LIN {X 0,Y 411.455,Z 725.231,A -85,B 0,C 180,E1 -10613.133,E2 -10613.133} C_VEL
LIN {X 0,Y 411.306,Z 725.25,A -85,B 0,C 180,E1 -10615.099,E2 -10615.099} C_VEL
LIN {X 0,Y 411.51,Z 725.225,A -85,B 0,C 180,E1 -10618.043,E2 -10618.043} C_VEL
LIN {X 0,Y 411.638,Z 725.209,A -85,B 0,C 180,E1 -10620,E2 -10620} C_VEL
LIN {X 0,Y 411.452,Z 725.232,A -85,B 0,C 180,E1 -10622.937,E2 -10622.937} C_VEL
LIN {X 0,Y 411.425,Z 725.236,A -85,B 0,C 180,E1 -10626.868,E2 -10626.868} C_VEL
LIN {X 0,Y 411.293,Z 725.251,A -85,B 0,C 180,E1 -10629.839,E2 -10629.839} C_VEL
LIN {X 0,Y 411.308,Z 725.25,A -85,B 0,C 180,E1 -10633.104,E2 -10633.104} C_VEL
LIN {X 0,Y 411.259,Z 725.258,A -85,B 0,C 180,E1 -10636.889,E2 -10636.889} C_VEL
LIN {X 0,Y 411.233,Z 725.259,A -85,B 0,C 180,E1 -10639.987,E2 -10639.987} C_VEL
LIN {X 0,Y 411.189,Z 725.266,A -85,B 0,C 180,E1 -10643.149,E2 -10643.149} C_VEL
LIN {X 0,Y 411.186,Z 725.265,A -85,B 0,C 180,E1 -10646.385,E2 -10646.385} C_VEL
LIN {X 0,Y 411.2,Z 725.264,A -85,B 0,C 180,E1 -10649.713,E2 -10649.713} C_VEL
LIN {X 0,Y 411.206,Z 725.265,A -85,B 0,C 180,E1 -10653.156,E2 -10653.156} C_VEL
LIN {X 0,Y 411.192,Z 725.264,A -85,B 0,C 180,E1 -10656.552,E2 -10656.552} C_VEL
LIN {X 0,Y 411.169,Z 725.268,A -85,B 0,C 180,E1 -10659.72,E2 -10659.72} C_VEL
LIN {X 0,Y 411.164,Z 725.268,A -85,B 0,C 180,E1 -10663.135,E2 -10663.135} C_VEL
LIN {X 0,Y 411.165,Z 725.268,A -85,B 0,C 180,E1 -10665.882,E2 -10665.882} C_VEL
LIN {X 0,Y 411.149,Z 725.27,A -85,B 0,C 180,E1 -10668.775,E2 -10668.775} C_VEL
LIN {X 0,Y 411.183,Z 725.266,A -85,B 0,C 180,E1 -10672.025,E2 -10672.025} C_VEL
LIN {X 0,Y 411.202,Z 725.263,A -85,B 0,C 180,E1 -10675.124,E2 -10675.124} C_VEL
LIN {X 0,Y 411.156,Z 725.269,A -85,B 0,C 180,E1 -10678.002,E2 -10678.002} C_VEL
LIN {X 0,Y 411.171,Z 725.267,A -85,B 0,C 180,E1 -10681.406,E2 -10681.406} C_VEL
LIN {X 0,Y 411.189,Z 725.267,A -85,B 0,C 180,E1 -10684.942,E2 -10684.942} C_VEL
LIN {X 0,Y 411.206,Z 725.263,A -85,B 0,C 180,E1 -10687.913,E2 -10687.913} C_VEL
LIN {X 0,Y 411.221,Z 725.263,A -85,B 0,C 180,E1 -10691.051,E2 -10691.051} C_VEL
LIN {X 0,Y 411.253,Z 725.258,A -85,B 0,C 180,E1 -10694.132,E2 -10694.132} C_VEL
LIN {X 0,Y 411.305,Z 725.253,A -85,B 0,C 180,E1 -10697.166,E2 -10697.166} C_VEL
LIN {X 0,Y 411.276,Z 725.254,A -85,B 0,C 180,E1 -10700.161,E2 -10700.161} C_VEL
LIN {X 0,Y 411.393,Z 725.242,A -85,B 0,C 180,E1 -10703.132,E2 -10703.132} C_VEL
LIN {X 0,Y 411.287,Z 725.254,A -85,B 0,C 180,E1 -10705.099,E2 -10705.099} C_VEL
LIN {X 0,Y 411.504,Z 725.224,A -85,B 0,C 180,E1 -10708.043,E2 -10708.043} C_VEL
LIN {X 0,Y 411.38,Z 725.241,A -85,B 0,C 180,E1 -10710.979,E2 -10710.979} C_VEL
LIN {X 0,Y 411.432,Z 725.234,A -85,B 0,C 180,E1 -10712.938,E2 -10712.938} C_VEL
LIN {X 0,Y 411.432,Z 725.235,A -85,B 0,C 180,E1 -10715.883,E2 -10715.883} C_VEL
LIN {X 0,Y 411.32,Z 725.247,A -85,B 0,C 180,E1 -10718.846,E2 -10718.846} C_VEL
LIN {X 0,Y 411.286,Z 725.255,A -85,B 0,C 180,E1 -10721.833,E2 -10721.833} C_VEL
LIN {X 0,Y 411.263,Z 725.254,A -85,B 0,C 180,E1 -10724.853,E2 -10724.853} C_VEL
LIN {X 0,Y 411.241,Z 725.258,A -85,B 0,C 180,E1 -10727.571,E2 -10727.571} C_VEL
LIN {X 0,Y 410.579,Z 725.344,A -85,B 0,C 180,E1 -10728.389,E2 -10728.389} C_VEL
LIN {X 0,Y 407.693,Z 725.704,A -85,B 0,C 180,E1 -10729.717,E2 -10729.717} C_VEL
LIN {X 0,Y 405.251,Z 726.005,A -85,B 0,C 180,E1 -10730.79,E2 -10730.79} C_VEL
LIN {X 0,Y 404.215,Z 726.134,A -85,B 0,C 180,E1 -10731.62,E2 -10731.62} C_VEL
LIN {X 0,Y 404.138,Z 726.14,A -85,B 0,C 180,E1 -10731.901,E2 -10731.901} C_VEL
LIN {X 0,Y 404.155,Z 726.139,A -85,B 0,C 180,E1 -10735.277,E2 -10735.277} C_VEL
LIN {X 0,Y 404.133,Z 726.147,A -85,B 0,C 180,E1 -10738.005,E2 -10738.005} C_VEL
LIN {X 0,Y 404.148,Z 726.143,A -85,B 0,C 180,E1 -10740.285,E2 -10740.285} C_VEL
LIN {X 0,Y 404.148,Z 726.142,A -85,B 0,C 180,E1 -10743.812,E2 -10743.812} C_VEL
LIN {X 0,Y 404.139,Z 726.141,A -85,B 0,C 180,E1 -10746.875,E2 -10746.875} C_VEL
LIN {X 0,Y 404.151,Z 726.142,A -85,B 0,C 180,E1 -10750.08,E2 -10750.08} C_VEL
LIN {X 0,Y 404.156,Z 726.139,A -85,B 0,C 180,E1 -10753.084,E2 -10753.084} C_VEL
LIN {X 0,Y 404.158,Z 726.14,A -85,B 0,C 180,E1 -10755.411,E2 -10755.411} C_VEL
LIN {X 0,Y 407.371,Z 737.515,A -85,B 0,C 180,E1 -10756.25,E2 -10756.25} C_VEL
LIN {X 0,Y 408.302,Z 740.837,A -85,B 0,C 180,E1 -10756.535,E2 -10756.535} C_VEL
LIN {X 0,Y 407.909,Z 751.917,A -85,B 0,C 180,E1 -10757.448,E2 -10757.448} C_VEL
LIN {X 0,Y 407.285,Z 762.487,A -85,B 0,C 180,E1 -10758.533,E2 -10758.533} C_VEL
LIN {X 0,Y 406.729,Z 771.783,A -85,B 0,C 180,E1 -10759.703,E2 -10759.703} C_VEL
LIN {X 0,Y 406.09,Z 781.183,A -85,B 0,C 180,E1 -10761.151,E2 -10761.151} C_VEL
LIN {X 0,Y 405.509,Z 789.001,A -85,B 0,C 180,E1 -10762.656,E2 -10762.656} C_VEL
LIN {X 0,Y 405.021,Z 795.844,A -85,B 0,C 180,E1 -10764.311,E2 -10764.311} C_VEL
LIN {X 0,Y 404.679,Z 800.21,A -85,B 0,C 180,E1 -10765.637,E2 -10765.637} C_VEL
LIN {X 0,Y 404.479,Z 804.684,A -85,B 0,C 180,E1 -10767.409,E2 -10767.409} C_VEL
LIN {X 0,Y 404.335,Z 806.818,A -85,B 0,C 180,E1 -10768.57,E2 -10768.57} C_VEL
LIN {X 0,Y 404.169,Z 809.071,A -85,B 0,C 180,E1 -10770.394,E2 -10770.394} C_VEL
LIN {X 0,Y 404.199,Z 809.968,A -85,B 0,C 180,E1 -10772.47,E2 -10772.47} C_VEL
LIN {X 0,Y 404.33,Z 809.377,A -85,B 0,C 180,E1 -10774.243,E2 -10774.243} C_VEL
LIN {X 0,Y 404.513,Z 808.375,A -85,B 0,C 180,E1 -10775.356,E2 -10775.356} C_VEL
LIN {X 0,Y 404.79,Z 806.008,A -85,B 0,C 180,E1 -10776.955,E2 -10776.955} C_VEL
LIN {X 0,Y 405.183,Z 802.282,A -85,B 0,C 180,E1 -10778.638,E2 -10778.638} C_VEL
LIN {X 0,Y 405.666,Z 797.413,A -85,B 0,C 180,E1 -10780.255,E2 -10780.255} C_VEL
LIN {X 0,Y 406.317,Z 791.148,A -85,B 0,C 180,E1 -10781.86,E2 -10781.86} C_VEL
LIN {X 0,Y 407.106,Z 783.159,A -85,B 0,C 180,E1 -10783.45,E2 -10783.45} C_VEL
LIN {X 0,Y 407.851,Z 774.76,A -85,B 0,C 180,E1 -10784.793,E2 -10784.793} C_VEL
LIN {X 0,Y 408.577,Z 764.958,A -85,B 0,C 180,E1 -10786.065,E2 -10786.065} C_VEL
LIN {X 0,Y 409.312,Z 753.636,A -85,B 0,C 180,E1 -10787.228,E2 -10787.228} C_VEL
LIN {X 0,Y 409.772,Z 744.554,A -85,B 0,C 180,E1 -10787.985,E2 -10787.985} C_VEL
LIN {X 0,Y 408.712,Z 739.651,A -85,B 0,C 180,E1 -10788.411,E2 -10788.411} C_VEL
LIN {X 0,Y 404.722,Z 727.908,A -85,B 0,C 180,E1 -10789.368,E2 -10789.368} C_VEL
LIN {X 0,Y 404.259,Z 726.133,A -85,B 0,C 180,E1 -10789.514,E2 -10789.514} C_VEL
LIN {X 0,Y 404.363,Z 726.114,A -85,B 0,C 180,E1 -10793.012,E2 -10793.012} C_VEL
LIN {X 0,Y 404.277,Z 726.124,A -85,B 0,C 180,E1 -10795.013,E2 -10795.013} C_VEL
LIN {X 0,Y 404.482,Z 726.104,A -85,B 0,C 180,E1 -10798.008,E2 -10798.008} C_VEL
LIN {X 0,Y 404.609,Z 726.087,A -85,B 0,C 180,E1 -10800,E2 -10800} C_VEL
LIN {X 0,Y 404.412,Z 726.103,A -85,B 0,C 180,E1 -10802.988,E2 -10802.988} C_VEL
LIN {X 0,Y 404.42,Z 726.105,A -85,B 0,C 180,E1 -10805.985,E2 -10805.985} C_VEL
LIN {X 0,Y 404.386,Z 726.112,A -85,B 0,C 180,E1 -10807.992,E2 -10807.992} C_VEL
LIN {X 0,Y 404.26,Z 726.125,A -85,B 0,C 180,E1 -10812.041,E2 -10812.041} C_VEL
LIN {X 0,Y 404.21,Z 726.127,A -85,B 0,C 180,E1 -10815.118,E2 -10815.118} C_VEL
LIN {X 0,Y 404.212,Z 726.132,A -85,B 0,C 180,E1 -10818.238,E2 -10818.238} C_VEL
LIN {X 0,Y 404.142,Z 726.137,A -85,B 0,C 180,E1 -10821.419,E2 -10821.419} C_VEL
LIN {X 0,Y 404.177,Z 726.14,A -85,B 0,C 180,E1 -10824.666,E2 -10824.666} C_VEL
LIN {X 0,Y 404.198,Z 726.138,A -85,B 0,C 180,E1 -10827.999,E2 -10827.999} C_VEL
LIN {X 0,Y 404.142,Z 726.141,A -85,B 0,C 180,E1 -10831.558,E2 -10831.558} C_VEL
LIN {X 0,Y 404.188,Z 726.138,A -85,B 0,C 180,E1 -10835.016,E2 -10835.016} C_VEL
LIN {X 0,Y 404.159,Z 726.145,A -85,B 0,C 180,E1 -10838.757,E2 -10838.757} C_VEL
LIN {X 0,Y 404.126,Z 726.148,A -85,B 0,C 180,E1 -10841.6,E2 -10841.6} C_VEL
LIN {X 0,Y 404.148,Z 726.144,A -85,B 0,C 180,E1 -10844.522,E2 -10844.522} C_VEL
LIN {X 0,Y 404.151,Z 726.237,A -85,B 0,C 180,E1 -10845.926,E2 -10845.926} C_VEL
LIN {X 0,Y 405.706,Z 733.429,A -85,B 0,C 180,E1 -10848.832,E2 -10848.832} C_VEL
LIN {X 0,Y 407.377,Z 742.456,A -85,B 0,C 180,E1 -10852.104,E2 -10852.104} C_VEL
LIN {X 0,Y 407.587,Z 746.68,A -85,B 0,C 180,E1 -10853.495,E2 -10853.495} C_VEL
LIN {X 0,Y 406.594,Z 758.282,A -85,B 0,C 180,E1 -10857.011,E2 -10857.011} C_VEL
LIN {X 0,Y 405.823,Z 768.597,A -85,B 0,C 180,E1 -10859.985,E2 -10859.985} C_VEL
LIN {X 0,Y 405.143,Z 781.14,A -85,B 0,C 180,E1 -10863.469,E2 -10863.469} C_VEL
LIN {X 0,Y 404.529,Z 794.458,A -85,B 0,C 180,E1 -10867.041,E2 -10867.041} C_VEL
LIN {X 0,Y 404.045,Z 806.932,A -85,B 0,C 180,E1 -10870.307,E2 -10870.307} C_VEL
LIN {X 0,Y 403.943,Z 812.973,A -85,B 0,C 180,E1 -10871.875,E2 -10871.875} C_VEL
LIN {X 0,Y 405.529,Z 827.395,A -85,B 0,C 180,E1 -10872.398,E2 -10872.398} C_VEL
LIN {X 0,Y 406.374,Z 841.524,A -85,B 0,C 180,E1 -10873.096,E2 -10873.096} C_VEL
LIN {X 0,Y 407.137,Z 852.896,A -85,B 0,C 180,E1 -10873.838,E2 -10873.838} C_VEL
LIN {X 0,Y 406.352,Z 864.193,A -85,B 0,C 180,E1 -10874.707,E2 -10874.707} C_VEL
LIN {X 0,Y 405.48,Z 875.869,A -85,B 0,C 180,E1 -10875.829,E2 -10875.829} C_VEL
LIN {X 0,Y 404.907,Z 885.404,A -85,B 0,C 180,E1 -10876.959,E2 -10876.959} C_VEL
LIN {X 0,Y 404.285,Z 894.164,A -85,B 0,C 180,E1 -10878.214,E2 -10878.214} C_VEL
LIN {X 0,Y 403.775,Z 902.798,A -85,B 0,C 180,E1 -10879.723,E2 -10879.723} C_VEL
LIN {X 0,Y 403.516,Z 909.827,A -85,B 0,C 180,E1 -10881.234,E2 -10881.234} C_VEL
LIN {X 0,Y 403.398,Z 916.317,A -85,B 0,C 180,E1 -10882.995,E2 -10882.995} C_VEL
LIN {X 0,Y 403.398,Z 920.58,A -85,B 0,C 180,E1 -10884.501,E2 -10884.501} C_VEL
LIN {X 0,Y 403.532,Z 923.776,A -85,B 0,C 180,E1 -10886.005,E2 -10886.005} C_VEL
LIN {X 0,Y 403.475,Z 926.402,A -85,B 0,C 180,E1 -10888.003,E2 -10888.003} C_VEL
LIN {X 0,Y 403.481,Z 927.104,A -85,B 0,C 180,E1 -10889.002,E2 -10889.002} C_VEL
LIN {X 0,Y 403.49,Z 927.365,A -85,B 0,C 180,E1 -10890,E2 -10890} C_VEL
LIN {X 0,Y 403.472,Z 927.18,A -85,B 0,C 180,E1 -10890.998,E2 -10890.998} C_VEL
LIN {X 0,Y 403.456,Z 926.592,A -85,B 0,C 180,E1 -10891.996,E2 -10891.996} C_VEL
LIN {X 0,Y 403.445,Z 925.596,A -85,B 0,C 180,E1 -10892.996,E2 -10892.996} C_VEL
LIN {X 0,Y 403.522,Z 924.151,A -85,B 0,C 180,E1 -10893.995,E2 -10893.995} C_VEL
LIN {X 0,Y 403.355,Z 921.099,A -85,B 0,C 180,E1 -10895.499,E2 -10895.499} C_VEL
LIN {X 0,Y 403.385,Z 916.972,A -85,B 0,C 180,E1 -10897.005,E2 -10897.005} C_VEL
LIN {X 0,Y 403.513,Z 910.613,A -85,B 0,C 180,E1 -10898.766,E2 -10898.766} C_VEL
LIN {X 0,Y 403.752,Z 903.688,A -85,B 0,C 180,E1 -10900.278,E2 -10900.278} C_VEL
LIN {X 0,Y 404.299,Z 895.087,A -85,B 0,C 180,E1 -10901.786,E2 -10901.786} C_VEL
LIN {X 0,Y 405.011,Z 886.285,A -85,B 0,C 180,E1 -10903.037,E2 -10903.037} C_VEL
LIN {X 0,Y 405.484,Z 877.813,A -85,B 0,C 180,E1 -10904.043,E2 -10904.043} C_VEL
LIN {X 0,Y 406.233,Z 866.186,A -85,B 0,C 180,E1 -10905.169,E2 -10905.169} C_VEL
LIN {X 0,Y 407.097,Z 854.815,A -85,B 0,C 180,E1 -10906.035,E2 -10906.035} C_VEL
LIN {X 0,Y 406.529,Z 845.674,A -85,B 0,C 180,E1 -10906.62,E2 -10906.62} C_VEL
LIN {X 0,Y 405.565,Z 832.566,A -85,B 0,C 180,E1 -10907.282,E2 -10907.282} C_VEL
LIN {X 0,Y 404.071,Z 818.692,A -85,B 0,C 180,E1 -10907.773,E2 -10907.773} C_VEL
LIN {X 0,Y 403.964,Z 816.966,A -85,B 0,C 180,E1 -10907.856,E2 -10907.856} C_VEL
LIN {X 0,Y 404.461,Z 803.727,A -85,B 0,C 180,E1 -10911.401,E2 -10911.401} C_VEL
LIN {X 0,Y 405.173,Z 790.061,A -85,B 0,C 180,E1 -10915.115,E2 -10915.115} C_VEL
LIN {X 0,Y 405.983,Z 778.085,A -85,B 0,C 180,E1 -10918.43,E2 -10918.43} C_VEL
LIN {X 0,Y 406.985,Z 764.176,A -85,B 0,C 180,E1 -10922.366,E2 -10922.366} C_VEL
LIN {X 0,Y 408.045,Z 752.225,A -85,B 0,C 180,E1 -10925.846,E2 -10925.846} C_VEL
LIN {X 0,Y 408.334,Z 748.205,A -85,B 0,C 180,E1 -10927.042,E2 -10927.042} C_VEL
LIN {X 0,Y 407.789,Z 744.091,A -85,B 0,C 180,E1 -10928.348,E2 -10928.348} C_VEL
LIN {X 0,Y 405.697,Z 733.602,A -85,B 0,C 180,E1 -10931.849,E2 -10931.849} C_VEL
LIN {X 0,Y 404.157,Z 726.141,A -85,B 0,C 180,E1 -10934.524,E2 -10934.524} C_VEL
LIN {X 0,Y 404.138,Z 726.145,A -85,B 0,C 180,E1 -10937.296,E2 -10937.296} C_VEL
LIN {X 0,Y 404.17,Z 726.138,A -85,B 0,C 180,E1 -10939.955,E2 -10939.955} C_VEL
LIN {X 0,Y 404.138,Z 726.142,A -85,B 0,C 180,E1 -10943.125,E2 -10943.125} C_VEL
LIN {X 0,Y 404.147,Z 726.141,A -85,B 0,C 180,E1 -10946.188,E2 -10946.188} C_VEL
LIN {X 0,Y 404.147,Z 726.146,A -85,B 0,C 180,E1 -10949.715,E2 -10949.715} C_VEL
LIN {X 0,Y 404.196,Z 726.134,A -85,B 0,C 180,E1 -10953.123,E2 -10953.123} C_VEL
LIN {X 0,Y 404.176,Z 726.137,A -85,B 0,C 180,E1 -10955.334,E2 -10955.334} C_VEL
LIN {X 0,Y 404.14,Z 726.142,A -85,B 0,C 180,E1 -10958.581,E2 -10958.581} C_VEL
LIN {X 0,Y 404.211,Z 726.135,A -85,B 0,C 180,E1 -10961.762,E2 -10961.762} C_VEL
LIN {X 0,Y 404.208,Z 726.133,A -85,B 0,C 180,E1 -10964.882,E2 -10964.882} C_VEL
LIN {X 0,Y 404.258,Z 726.13,A -85,B 0,C 180,E1 -10967.959,E2 -10967.959} C_VEL
LIN {X 0,Y 404.407,Z 726.112,A -85,B 0,C 180,E1 -10972.129,E2 -10972.129} C_VEL
LIN {X 0,Y 404.422,Z 726.108,A -85,B 0,C 180,E1 -10974.015,E2 -10974.015} C_VEL
LIN {X 0,Y 404.479,Z 726.101,A -85,B 0,C 180,E1 -10978.009,E2 -10978.009} C_VEL
LIN {X 0,Y 404.608,Z 726.084,A -85,B 0,C 180,E1 -10980,E2 -10980} C_VEL
LIN {X 0,Y 404.41,Z 726.109,A -85,B 0,C 180,E1 -10982.989,E2 -10982.989} C_VEL
LIN {X 0,Y 404.371,Z 726.115,A -85,B 0,C 180,E1 -10986.988,E2 -10986.988} C_VEL
LIN {X 0,Y 404.259,Z 726.127,A -85,B 0,C 180,E1 -10990.012,E2 -10990.012} C_VEL
LIN {X 0,Y 404.269,Z 726.127,A -85,B 0,C 180,E1 -10993.211,E2 -10993.211} C_VEL
LIN {X 0,Y 404.218,Z 726.135,A -85,B 0,C 180,E1 -10997.007,E2 -10997.007} C_VEL
LIN {X 0,Y 404.166,Z 726.139,A -85,B 0,C 180,E1 -11000.352,E2 -11000.352} C_VEL
LIN {X 0,Y 404.15,Z 726.142,A -85,B 0,C 180,E1 -11003.576,E2 -11003.576} C_VEL
LIN {X 0,Y 404.131,Z 726.145,A -85,B 0,C 180,E1 -11006.882,E2 -11006.882} C_VEL
LIN {X 0,Y 404.146,Z 726.142,A -85,B 0,C 180,E1 -11010.285,E2 -11010.285} C_VEL
LIN {X 0,Y 404.14,Z 726.144,A -85,B 0,C 180,E1 -11013.813,E2 -11013.813} C_VEL
LIN {X 0,Y 404.135,Z 726.143,A -85,B 0,C 180,E1 -11016.874,E2 -11016.874} C_VEL
LIN {X 0,Y 404.118,Z 726.147,A -85,B 0,C 180,E1 -11020.075,E2 -11020.075} C_VEL
LIN {X 0,Y 404.143,Z 726.142,A -85,B 0,C 180,E1 -11023.082,E2 -11023.082} C_VEL
LIN {X 0,Y 404.122,Z 726.146,A -85,B 0,C 180,E1 -11025.922,E2 -11025.922} C_VEL
LIN {X 0,Y 404.103,Z 726.148,A -85,B 0,C 180,E1 -11028.633,E2 -11028.633} C_VEL
LIN {X 0,Y 404.139,Z 726.144,A -85,B 0,C 180,E1 -11031.495,E2 -11031.495} C_VEL
LIN {X 0,Y 404.173,Z 726.138,A -85,B 0,C 180,E1 -11034.983,E2 -11034.983} C_VEL
LIN {X 0,Y 404.133,Z 726.145,A -85,B 0,C 180,E1 -11038.444,E2 -11038.444} C_VEL
LIN {X 0,Y 404.15,Z 726.143,A -85,B 0,C 180,E1 -11040.862,E2 -11040.862} C_VEL
LIN {X 0,Y 404.153,Z 726.143,A -85,B 0,C 180,E1 -11044.723,E2 -11044.723} C_VEL
LIN {X 0,Y 404.168,Z 726.138,A -85,B 0,C 180,E1 -11047.508,E2 -11047.508} C_VEL
LIN {X 0,Y 404.165,Z 726.141,A -85,B 0,C 180,E1 -11050.708,E2 -11050.708} C_VEL
LIN {X 0,Y 404.221,Z 726.132,A -85,B 0,C 180,E1 -11053.848,E2 -11053.848} C_VEL
LIN {X 0,Y 404.286,Z 726.127,A -85,B 0,C 180,E1 -11056.939,E2 -11056.939} C_VEL
LIN {X 0,Y 404.244,Z 726.129,A -85,B 0,C 180,E1 -11059.988,E2 -11059.988} C_VEL
LIN {X 0,Y 404.343,Z 726.119,A -85,B 0,C 180,E1 -11063.012,E2 -11063.012} C_VEL
LIN {X 0,Y 404.259,Z 726.129,A -85,B 0,C 180,E1 -11065.013,E2 -11065.013} C_VEL
LIN {X 0,Y 404.473,Z 726.1,A -85,B 0,C 180,E1 -11068.009,E2 -11068.009} C_VEL
LIN {X 0,Y 404.35,Z 726.117,A -85,B 0,C 180,E1 -11070.996,E2 -11070.996} C_VEL
LIN {X 0,Y 404.392,Z 726.112,A -85,B 0,C 180,E1 -11072.989,E2 -11072.989} C_VEL
LIN {X 0,Y 404.381,Z 726.112,A -85,B 0,C 180,E1 -11075.986,E2 -11075.986} C_VEL
LIN {X 0,Y 404.268,Z 726.126,A -85,B 0,C 180,E1 -11079.002,E2 -11079.002} C_VEL
LIN {X 0,Y 404.259,Z 726.128,A -85,B 0,C 180,E1 -11082.042,E2 -11082.042} C_VEL
LIN {X 0,Y 404.209,Z 726.133,A -85,B 0,C 180,E1 -11085.118,E2 -11085.118} C_VEL
LIN {X 0,Y 404.212,Z 726.133,A -85,B 0,C 180,E1 -11088.238,E2 -11088.238} C_VEL
LIN {X 0,Y 404.142,Z 726.142,A -85,B 0,C 180,E1 -11091.419,E2 -11091.419} C_VEL
LIN {X 0,Y 404.138,Z 726.14,A -85,B 0,C 180,E1 -11091.901,E2 -11091.901} C_VEL
LIN {X 0,Y 403.496,Z 726.222,A -85,B 0,C 180,E1 -11092.733,E2 -11092.733} C_VEL
LIN {X 0,Y 400.668,Z 726.579,A -85,B 0,C 180,E1 -11094.084,E2 -11094.084} C_VEL
LIN {X 0,Y 398.249,Z 726.883,A -85,B 0,C 180,E1 -11095.176,E2 -11095.176} C_VEL
LIN {X 0,Y 397.191,Z 727.012,A -85,B 0,C 180,E1 -11096.019,E2 -11096.019} C_VEL
LIN {X 0,Y 397.095,Z 727.021,A -85,B 0,C 180,E1 -11096.305,E2 -11096.305} C_VEL
LIN {X 0,Y 397.104,Z 727.021,A -85,B 0,C 180,E1 -11099.863,E2 -11099.863} C_VEL
LIN {X 0,Y 397.122,Z 727.016,A -85,B 0,C 180,E1 -11103.718,E2 -11103.718} C_VEL
LIN {X 0,Y 397.096,Z 727.017,A -85,B 0,C 180,E1 -11107.209,E2 -11107.209} C_VEL
LIN {X 0,Y 397.105,Z 727.022,A -85,B 0,C 180,E1 -11110.445,E2 -11110.445} C_VEL
LIN {X 0,Y 397.104,Z 727.017,A -85,B 0,C 180,E1 -11113.649,E2 -11113.649} C_VEL
LIN {X 0,Y 397.111,Z 727.023,A -85,B 0,C 180,E1 -11115.156,E2 -11115.156} C_VEL
LIN {X 0,Y 400.422,Z 738.626,A -85,B 0,C 180,E1 -11116.023,E2 -11116.023} C_VEL
LIN {X 0,Y 401.529,Z 743.37,A -85,B 0,C 180,E1 -11116.427,E2 -11116.427} C_VEL
LIN {X 0,Y 400.921,Z 754.73,A -85,B 0,C 180,E1 -11117.413,E2 -11117.413} C_VEL
LIN {X 0,Y 400.248,Z 766.257,A -85,B 0,C 180,E1 -11118.67,E2 -11118.67} C_VEL
LIN {X 0,Y 399.555,Z 776.377,A -85,B 0,C 180,E1 -11120.057,E2 -11120.057} C_VEL
LIN {X 0,Y 398.874,Z 785.472,A -85,B 0,C 180,E1 -11121.604,E2 -11121.604} C_VEL
LIN {X 0,Y 398.368,Z 792.688,A -85,B 0,C 180,E1 -11123.142,E2 -11123.142} C_VEL
LIN {X 0,Y 397.823,Z 799.388,A -85,B 0,C 180,E1 -11124.96,E2 -11124.96} C_VEL
LIN {X 0,Y 397.54,Z 804.385,A -85,B 0,C 180,E1 -11126.767,E2 -11126.767} C_VEL
LIN {X 0,Y 397.391,Z 807.1,A -85,B 0,C 180,E1 -11128.093,E2 -11128.093} C_VEL
LIN {X 0,Y 397.244,Z 808.728,A -85,B 0,C 180,E1 -11129.132,E2 -11129.132} C_VEL
LIN {X 0,Y 397.158,Z 810.018,A -85,B 0,C 180,E1 -11130.298,E2 -11130.298} C_VEL
LIN {X 0,Y 397.179,Z 811.029,A -85,B 0,C 180,E1 -11132.22,E2 -11132.22} C_VEL
LIN {X 0,Y 397.27,Z 810.791,A -85,B 0,C 180,E1 -11133.751,E2 -11133.751} C_VEL
LIN {X 0,Y 397.42,Z 810.005,A -85,B 0,C 180,E1 -11134.886,E2 -11134.886} C_VEL
LIN {X 0,Y 397.759,Z 807.642,A -85,B 0,C 180,E1 -11136.75,E2 -11136.75} C_VEL
LIN {X 0,Y 398.107,Z 804.708,A -85,B 0,C 180,E1 -11138.239,E2 -11138.239} C_VEL
LIN {X 0,Y 398.553,Z 800.302,A -85,B 0,C 180,E1 -11139.888,E2 -11139.888} C_VEL
LIN {X 0,Y 399.253,Z 794.484,A -85,B 0,C 180,E1 -11141.527,E2 -11141.527} C_VEL
LIN {X 0,Y 399.998,Z 787.113,A -85,B 0,C 180,E1 -11143.147,E2 -11143.147} C_VEL
LIN {X 0,Y 400.827,Z 778.512,A -85,B 0,C 180,E1 -11144.658,E2 -11144.658} C_VEL
LIN {X 0,Y 401.637,Z 769.297,A -85,B 0,C 180,E1 -11145.949,E2 -11145.949} C_VEL
LIN {X 0,Y 402.39,Z 758.629,A -85,B 0,C 180,E1 -11147.159,E2 -11147.159} C_VEL
LIN {X 0,Y 403.017,Z 748.139,A -85,B 0,C 180,E1 -11148.11,E2 -11148.11} C_VEL
LIN {X 0,Y 403.101,Z 745.629,A -85,B 0,C 180,E1 -11148.306,E2 -11148.306} C_VEL
LIN {X 0,Y 400.551,Z 736.775,A -85,B 0,C 180,E1 -11149.102,E2 -11149.102} C_VEL
LIN {X 0,Y 397.21,Z 727.012,A -85,B 0,C 180,E1 -11149.873,E2 -11149.873} C_VEL
LIN {X 0,Y 397.309,Z 726.993,A -85,B 0,C 180,E1 -11152.887,E2 -11152.887} C_VEL
LIN {X 0,Y 397.247,Z 727,A -85,B 0,C 180,E1 -11154.925,E2 -11154.925} C_VEL
LIN {X 0,Y 397.451,Z 726.98,A -85,B 0,C 180,E1 -11157.973,E2 -11157.973} C_VEL
LIN {X 0,Y 397.579,Z 726.962,A -85,B 0,C 180,E1 -11160,E2 -11160} C_VEL
LIN {X 0,Y 397.372,Z 726.98,A -85,B 0,C 180,E1 -11163.041,E2 -11163.041} C_VEL
LIN {X 0,Y 397.371,Z 726.983,A -85,B 0,C 180,E1 -11166.091,E2 -11166.091} C_VEL
LIN {X 0,Y 397.331,Z 726.989,A -85,B 0,C 180,E1 -11168.135,E2 -11168.135} C_VEL
LIN {X 0,Y 397.202,Z 727.005,A -85,B 0,C 180,E1 -11171.223,E2 -11171.223} C_VEL
LIN {X 0,Y 397.18,Z 727.007,A -85,B 0,C 180,E1 -11174.343,E2 -11174.343} C_VEL
LIN {X 0,Y 397.177,Z 727.01,A -85,B 0,C 180,E1 -11177.506,E2 -11177.506} C_VEL
LIN {X 0,Y 397.106,Z 727.014,A -85,B 0,C 180,E1 -11180.73,E2 -11180.73} C_VEL
LIN {X 0,Y 397.132,Z 727.013,A -85,B 0,C 180,E1 -11184.018,E2 -11184.018} C_VEL
LIN {X 0,Y 397.197,Z 727.007,A -85,B 0,C 180,E1 -11187.39,E2 -11187.39} C_VEL
LIN {X 0,Y 397.081,Z 727.02,A -85,B 0,C 180,E1 -11190.882,E2 -11190.882} C_VEL
LIN {X 0,Y 397.128,Z 727.02,A -85,B 0,C 180,E1 -11194.493,E2 -11194.493} C_VEL
LIN {X 0,Y 397.106,Z 727.025,A -85,B 0,C 180,E1 -11198.275,E2 -11198.275} C_VEL
LIN {X 0,Y 397.091,Z 727.028,A -85,B 0,C 180,E1 -11200.909,E2 -11200.909} C_VEL
LIN {X 0,Y 397.104,Z 727.023,A -85,B 0,C 180,E1 -11203.648,E2 -11203.648} C_VEL
LIN {X 0,Y 397.115,Z 727.126,A -85,B 0,C 180,E1 -11205.418,E2 -11205.418} C_VEL
LIN {X 0,Y 398.691,Z 734.52,A -85,B 0,C 180,E1 -11208.518,E2 -11208.518} C_VEL
LIN {X 0,Y 400.16,Z 742.261,A -85,B 0,C 180,E1 -11211.428,E2 -11211.428} C_VEL
LIN {X 0,Y 400.702,Z 746.125,A -85,B 0,C 180,E1 -11212.784,E2 -11212.784} C_VEL
LIN {X 0,Y 400.114,Z 753.694,A -85,B 0,C 180,E1 -11215.19,E2 -11215.19} C_VEL
LIN {X 0,Y 399.305,Z 763.407,A -85,B 0,C 180,E1 -11218.128,E2 -11218.128} C_VEL
LIN {X 0,Y 398.345,Z 777.857,A -85,B 0,C 180,E1 -11222.29,E2 -11222.29} C_VEL
LIN {X 0,Y 397.67,Z 790.287,A -85,B 0,C 180,E1 -11225.739,E2 -11225.739} C_VEL
LIN {X 0,Y 397.119,Z 803.372,A -85,B 0,C 180,E1 -11229.271,E2 -11229.271} C_VEL
LIN {X 0,Y 396.9,Z 811.706,A -85,B 0,C 180,E1 -11231.478,E2 -11231.478} C_VEL
LIN {X 0,Y 398.69,Z 827.102,A -85,B 0,C 180,E1 -11232.074,E2 -11232.074} C_VEL
LIN {X 0,Y 399.384,Z 839.916,A -85,B 0,C 180,E1 -11232.725,E2 -11232.725} C_VEL
LIN {X 0,Y 399.931,Z 850.348,A -85,B 0,C 180,E1 -11233.407,E2 -11233.407} C_VEL
LIN {X 0,Y 400.075,Z 855.666,A -85,B 0,C 180,E1 -11233.807,E2 -11233.807} C_VEL
LIN {X 0,Y 399.105,Z 867.483,A -85,B 0,C 180,E1 -11234.815,E2 -11234.815} C_VEL
LIN {X 0,Y 398.339,Z 877.828,A -85,B 0,C 180,E1 -11235.906,E2 -11235.906} C_VEL
LIN {X 0,Y 397.887,Z 884.445,A -85,B 0,C 180,E1 -11236.725,E2 -11236.725} C_VEL
LIN {X 0,Y 397.165,Z 894.743,A -85,B 0,C 180,E1 -11238.258,E2 -11238.258} C_VEL
LIN {X 0,Y 396.67,Z 903.114,A -85,B 0,C 180,E1 -11239.795,E2 -11239.795} C_VEL
LIN {X 0,Y 396.417,Z 909.875,A -85,B 0,C 180,E1 -11241.333,E2 -11241.333} C_VEL
LIN {X 0,Y 396.323,Z 916.429,A -85,B 0,C 180,E1 -11243.241,E2 -11243.241} C_VEL
LIN {X 0,Y 396.399,Z 920.741,A -85,B 0,C 180,E1 -11244.914,E2 -11244.914} C_VEL
LIN {X 0,Y 396.478,Z 922.753,A -85,B 0,C 180,E1 -11245.934,E2 -11245.934} C_VEL
LIN {X 0,Y 396.425,Z 924.273,A -85,B 0,C 180,E1 -11246.951,E2 -11246.951} C_VEL
LIN {X 0,Y 396.438,Z 925.387,A -85,B 0,C 180,E1 -11247.968,E2 -11247.968} C_VEL
LIN {X 0,Y 396.45,Z 926.09,A -85,B 0,C 180,E1 -11248.984,E2 -11248.984} C_VEL
LIN {X 0,Y 396.464,Z 926.345,A -85,B 0,C 180,E1 -11250,E2 -11250} C_VEL
LIN {X 0,Y 396.442,Z 926.161,A -85,B 0,C 180,E1 -11251.016,E2 -11251.016} C_VEL
LIN {X 0,Y 396.42,Z 925.57,A -85,B 0,C 180,E1 -11252.032,E2 -11252.032} C_VEL
LIN {X 0,Y 396.409,Z 924.57,A -85,B 0,C 180,E1 -11253.049,E2 -11253.049} C_VEL
LIN {X 0,Y 396.487,Z 923.112,A -85,B 0,C 180,E1 -11254.066,E2 -11254.066} C_VEL
LIN {X 0,Y 396.294,Z 920.045,A -85,B 0,C 180,E1 -11255.597,E2 -11255.597} C_VEL
LIN {X 0,Y 396.311,Z 915.902,A -85,B 0,C 180,E1 -11257.131,E2 -11257.131} C_VEL
LIN {X 0,Y 396.432,Z 909.526,A -85,B 0,C 180,E1 -11258.924,E2 -11258.924} C_VEL
LIN {X 0,Y 396.714,Z 902.585,A -85,B 0,C 180,E1 -11260.462,E2 -11260.462} C_VEL
LIN {X 0,Y 397.269,Z 893.944,A -85,B 0,C 180,E1 -11261.997,E2 -11261.997} C_VEL
LIN {X 0,Y 397.979,Z 885.102,A -85,B 0,C 180,E1 -11263.272,E2 -11263.272} C_VEL
LIN {X 0,Y 398.574,Z 875.408,A -85,B 0,C 180,E1 -11264.422,E2 -11264.422} C_VEL
LIN {X 0,Y 399.39,Z 864.918,A -85,B 0,C 180,E1 -11265.435,E2 -11265.435} C_VEL
LIN {X 0,Y 400.165,Z 853.403,A -85,B 0,C 180,E1 -11266.32,E2 -11266.32} C_VEL
LIN {X 0,Y 399.159,Z 840.394,A -85,B 0,C 180,E1 -11267.131,E2 -11267.131} C_VEL
LIN {X 0,Y 398.138,Z 828.268,A -85,B 0,C 180,E1 -11267.701,E2 -11267.701} C_VEL
LIN {X 0,Y 396.89,Z 816.157,A -85,B 0,C 180,E1 -11268.118,E2 -11268.118} C_VEL
LIN {X 0,Y 397.445,Z 802.734,A -85,B 0,C 180,E1 -11271.798,E2 -11271.798} C_VEL
LIN {X 0,Y 398.206,Z 789.582,A -85,B 0,C 180,E1 -11275.457,E2 -11275.457} C_VEL
LIN {X 0,Y 399.042,Z 777.162,A -85,B 0,C 180,E1 -11278.969,E2 -11278.969} C_VEL
LIN {X 0,Y 400.175,Z 763.287,A -85,B 0,C 180,E1 -11282.986,E2 -11282.986} C_VEL
LIN {X 0,Y 401.298,Z 751.355,A -85,B 0,C 180,E1 -11286.545,E2 -11286.545} C_VEL
LIN {X 0,Y 401.14,Z 746.836,A -85,B 0,C 180,E1 -11287.963,E2 -11287.963} C_VEL
LIN {X 0,Y 399.005,Z 736.307,A -85,B 0,C 180,E1 -11291.515,E2 -11291.515} C_VEL
LIN {X 0,Y 397.111,Z 727.02,A -85,B 0,C 180,E1 -11294.845,E2 -11294.845} C_VEL
LIN {X 0,Y 397.068,Z 727.025,A -85,B 0,C 180,E1 -11298.021,E2 -11298.021} C_VEL
LIN {X 0,Y 397.131,Z 727.017,A -85,B 0,C 180,E1 -11301.139,E2 -11301.139} C_VEL
LIN {X 0,Y 397.121,Z 727.015,A -85,B 0,C 180,E1 -11304.497,E2 -11304.497} C_VEL
LIN {X 0,Y 397.08,Z 727.023,A -85,B 0,C 180,E1 -11307.929,E2 -11307.929} C_VEL
LIN {X 0,Y 397.124,Z 727.017,A -85,B 0,C 180,E1 -11311.456,E2 -11311.456} C_VEL
LIN {X 0,Y 397.154,Z 727.012,A -85,B 0,C 180,E1 -11314.488,E2 -11314.488} C_VEL
LIN {X 0,Y 397.098,Z 727.021,A -85,B 0,C 180,E1 -11318.182,E2 -11318.182} C_VEL
LIN {X 0,Y 397.163,Z 727.01,A -85,B 0,C 180,E1 -11321.427,E2 -11321.427} C_VEL
LIN {X 0,Y 397.181,Z 727.009,A -85,B 0,C 180,E1 -11324.608,E2 -11324.608} C_VEL
LIN {X 0,Y 397.221,Z 727.004,A -85,B 0,C 180,E1 -11327.742,E2 -11327.742} C_VEL
LIN {X 0,Y 397.255,Z 727,A -85,B 0,C 180,E1 -11330.838,E2 -11330.838} C_VEL
LIN {X 0,Y 397.373,Z 726.985,A -85,B 0,C 180,E1 -11333.909,E2 -11333.909} C_VEL
LIN {X 0,Y 397.448,Z 726.976,A -85,B 0,C 180,E1 -11337.973,E2 -11337.973} C_VEL
LIN {X 0,Y 397.577,Z 726.96,A -85,B 0,C 180,E1 -11340,E2 -11340} C_VEL
LIN {X 0,Y 397.369,Z 726.986,A -85,B 0,C 180,E1 -11343.042,E2 -11343.042} C_VEL
LIN {X 0,Y 397.319,Z 726.99,A -85,B 0,C 180,E1 -11346.521,E2 -11346.521} C_VEL
LIN {X 0,Y 397.238,Z 727.003,A -85,B 0,C 180,E1 -11349.162,E2 -11349.162} C_VEL
LIN {X 0,Y 397.221,Z 727.004,A -85,B 0,C 180,E1 -11352.258,E2 -11352.258} C_VEL
LIN {X 0,Y 397.18,Z 727.01,A -85,B 0,C 180,E1 -11355.392,E2 -11355.392} C_VEL
LIN {X 0,Y 397.16,Z 727.012,A -85,B 0,C 180,E1 -11358.574,E2 -11358.574} C_VEL
LIN {X 0,Y 397.097,Z 727.021,A -85,B 0,C 180,E1 -11361.819,E2 -11361.819} C_VEL
LIN {X 0,Y 397.099,Z 727.022,A -85,B 0,C 180,E1 -11365.136,E2 -11365.136} C_VEL
LIN {X 0,Y 397.079,Z 727.022,A -85,B 0,C 180,E1 -11368.547,E2 -11368.547} C_VEL
LIN {X 0,Y 397.083,Z 727.023,A -85,B 0,C 180,E1 -11371.836,E2 -11371.836} C_VEL
LIN {X 0,Y 397.119,Z 727.017,A -85,B 0,C 180,E1 -11374.494,E2 -11374.494} C_VEL
LIN {X 0,Y 397.092,Z 727.022,A -85,B 0,C 180,E1 -11378.277,E2 -11378.277} C_VEL
LIN {X 0,Y 397.053,Z 727.027,A -85,B 0,C 180,E1 -11381.977,E2 -11381.977} C_VEL
LIN {X 0,Y 397.086,Z 727.021,A -85,B 0,C 180,E1 -11385.069,E2 -11385.069} C_VEL
LIN {X 0,Y 397.053,Z 727.027,A -85,B 0,C 180,E1 -11388.024,E2 -11388.024} C_VEL
LIN {X 0,Y 397.091,Z 727.023,A -85,B 0,C 180,E1 -11391.724,E2 -11391.724} C_VEL
LIN {X 0,Y 397.117,Z 727.018,A -85,B 0,C 180,E1 -11395.506,E2 -11395.506} C_VEL
LIN {X 0,Y 397.073,Z 727.023,A -85,B 0,C 180,E1 -11399.117,E2 -11399.117} C_VEL
LIN {X 0,Y 397.06,Z 727.026,A -85,B 0,C 180,E1 -11402.253,E2 -11402.253} C_VEL
LIN {X 0,Y 397.103,Z 727.021,A -85,B 0,C 180,E1 -11404.865,E2 -11404.865} C_VEL
LIN {X 0,Y 397.097,Z 727.021,A -85,B 0,C 180,E1 -11408.182,E2 -11408.182} C_VEL
LIN {X 0,Y 397.16,Z 727.012,A -85,B 0,C 180,E1 -11411.426,E2 -11411.426} C_VEL
LIN {X 0,Y 397.178,Z 727.011,A -85,B 0,C 180,E1 -11414.608,E2 -11414.608} C_VEL
LIN {X 0,Y 397.216,Z 727.004,A -85,B 0,C 180,E1 -11417.742,E2 -11417.742} C_VEL
LIN {X 0,Y 397.229,Z 727.005,A -85,B 0,C 180,E1 -11420.838,E2 -11420.838} C_VEL
LIN {X 0,Y 397.323,Z 726.991,A -85,B 0,C 180,E1 -11423.908,E2 -11423.908} C_VEL
LIN {X 0,Y 397.442,Z 726.976,A -85,B 0,C 180,E1 -11427.973,E2 -11427.973} C_VEL
LIN {X 0,Y 397.443,Z 726.976,A -85,B 0,C 180,E1 -11432.027,E2 -11432.027} C_VEL
LIN {X 0,Y 397.332,Z 726.99,A -85,B 0,C 180,E1 -11436.092,E2 -11436.092} C_VEL
LIN {X 0,Y 397.238,Z 727.003,A -85,B 0,C 180,E1 -11439.162,E2 -11439.162} C_VEL
LIN {X 0,Y 397.222,Z 727.003,A -85,B 0,C 180,E1 -11442.258,E2 -11442.258} C_VEL
LIN {X 0,Y 397.182,Z 727.01,A -85,B 0,C 180,E1 -11445.392,E2 -11445.392} C_VEL
LIN {X 0,Y 397.164,Z 727.01,A -85,B 0,C 180,E1 -11448.574,E2 -11448.574} C_VEL
LIN {X 0,Y 397.095,Z 727.022,A -85,B 0,C 180,E1 -11451.894,E2 -11451.894} C_VEL
LIN {X 0,Y 397.11,Z 727.017,A -85,B 0,C 180,E1 -11455.135,E2 -11455.135} C_VEL
LIN {X 0,Y 397.095,Z 727.021,A -85,B 0,C 180,E1 -11456.305,E2 -11456.305} C_VEL
LIN {X 0,Y 396.402,Z 727.105,A -85,B 0,C 180,E1 -11457.152,E2 -11457.152} C_VEL
LIN {X 0,Y 393.544,Z 727.462,A -85,B 0,C 180,E1 -11458.529,E2 -11458.529} C_VEL
LIN {X 0,Y 391.137,Z 727.762,A -85,B 0,C 180,E1 -11459.641,E2 -11459.641} C_VEL
LIN {X 0,Y 390.101,Z 727.892,A -85,B 0,C 180,E1 -11460.5,E2 -11460.5} C_VEL
LIN {X 0,Y 390.014,Z 727.9,A -85,B 0,C 180,E1 -11460.792,E2 -11460.792} C_VEL
LIN {X 0,Y 390.071,Z 727.897,A -85,B 0,C 180,E1 -11464.025,E2 -11464.025} C_VEL
LIN {X 0,Y 390.045,Z 727.896,A -85,B 0,C 180,E1 -11467.551,E2 -11467.551} C_VEL
LIN {X 0,Y 390.059,Z 727.895,A -85,B 0,C 180,E1 -11470.821,E2 -11470.821} C_VEL
LIN {X 0,Y 390.059,Z 727.895,A -85,B 0,C 180,E1 -11473.886,E2 -11473.886} C_VEL
LIN {X 0,Y 390.068,Z 727.898,A -85,B 0,C 180,E1 -11474.89,E2 -11474.89} C_VEL
LIN {X 0,Y 393.471,Z 739.805,A -85,B 0,C 180,E1 -11475.801,E2 -11475.801} C_VEL
LIN {X 0,Y 394.567,Z 743.975,A -85,B 0,C 180,E1 -11476.169,E2 -11476.169} C_VEL
LIN {X 0,Y 394.062,Z 755.61,A -85,B 0,C 180,E1 -11477.197,E2 -11477.197} C_VEL
LIN {X 0,Y 393.349,Z 766.933,A -85,B 0,C 180,E1 -11478.446,E2 -11478.446} C_VEL
LIN {X 0,Y 392.719,Z 776.261,A -85,B 0,C 180,E1 -11479.723,E2 -11479.723} C_VEL
LIN {X 0,Y 392.051,Z 784.714,A -85,B 0,C 180,E1 -11481.14,E2 -11481.14} C_VEL
LIN {X 0,Y 391.489,Z 792.308,A -85,B 0,C 180,E1 -11482.708,E2 -11482.708} C_VEL
LIN {X 0,Y 390.984,Z 798.896,A -85,B 0,C 180,E1 -11484.417,E2 -11484.417} C_VEL
LIN {X 0,Y 390.581,Z 803.877,A -85,B 0,C 180,E1 -11486.096,E2 -11486.096} C_VEL
LIN {X 0,Y 390.408,Z 807.613,A -85,B 0,C 180,E1 -11487.788,E2 -11487.788} C_VEL
LIN {X 0,Y 390.18,Z 810.629,A -85,B 0,C 180,E1 -11489.836,E2 -11489.836} C_VEL
LIN {X 0,Y 390.129,Z 811.516,A -85,B 0,C 180,E1 -11490.896,E2 -11490.896} C_VEL
LIN {X 0,Y 390.156,Z 812.039,A -85,B 0,C 180,E1 -11492.073,E2 -11492.073} C_VEL
LIN {X 0,Y 390.209,Z 812.04,A -85,B 0,C 180,E1 -11493.239,E2 -11493.239} C_VEL
LIN {X 0,Y 390.369,Z 811.517,A -85,B 0,C 180,E1 -11494.4,E2 -11494.4} C_VEL
LIN {X 0,Y 390.525,Z 810.54,A -85,B 0,C 180,E1 -11495.549,E2 -11495.549} C_VEL
LIN {X 0,Y 390.771,Z 809.004,A -85,B 0,C 180,E1 -11496.692,E2 -11496.692} C_VEL
LIN {X 0,Y 391.159,Z 805.802,A -85,B 0,C 180,E1 -11498.387,E2 -11498.387} C_VEL
LIN {X 0,Y 391.642,Z 801.409,A -85,B 0,C 180,E1 -11500.065,E2 -11500.065} C_VEL
LIN {X 0,Y 392.436,Z 795.108,A -85,B 0,C 180,E1 -11501.857,E2 -11501.857} C_VEL
LIN {X 0,Y 393.2,Z 788.257,A -85,B 0,C 180,E1 -11503.382,E2 -11503.382} C_VEL
LIN {X 0,Y 394.05,Z 779.897,A -85,B 0,C 180,E1 -11504.881,E2 -11504.881} C_VEL
LIN {X 0,Y 394.928,Z 770.458,A -85,B 0,C 180,E1 -11506.23,E2 -11506.23} C_VEL
LIN {X 0,Y 395.726,Z 759.798,A -85,B 0,C 180,E1 -11507.461,E2 -11507.461} C_VEL
LIN {X 0,Y 396.416,Z 748.766,A -85,B 0,C 180,E1 -11508.472,E2 -11508.472} C_VEL
LIN {X 0,Y 396.467,Z 747.409,A -85,B 0,C 180,E1 -11508.579,E2 -11508.579} C_VEL
LIN {X 0,Y 393.547,Z 737.539,A -85,B 0,C 180,E1 -11509.502,E2 -11509.502} C_VEL
LIN {X 0,Y 390.188,Z 727.883,A -85,B 0,C 180,E1 -11510.311,E2 -11510.311} C_VEL
LIN {X 0,Y 390.298,Z 727.867,A -85,B 0,C 180,E1 -11513.797,E2 -11513.797} C_VEL
LIN {X 0,Y 390.419,Z 727.856,A -85,B 0,C 180,E1 -11517.937,E2 -11517.937} C_VEL
LIN {X 0,Y 390.548,Z 727.838,A -85,B 0,C 180,E1 -11520,E2 -11520} C_VEL
LIN {X 0,Y 390.306,Z 727.86,A -85,B 0,C 180,E1 -11523.096,E2 -11523.096} C_VEL
LIN {X 0,Y 390.324,Z 727.861,A -85,B 0,C 180,E1 -11526.202,E2 -11526.202} C_VEL
LIN {X 0,Y 390.201,Z 727.872,A -85,B 0,C 180,E1 -11529.329,E2 -11529.329} C_VEL
LIN {X 0,Y 390.174,Z 727.88,A -85,B 0,C 180,E1 -11532.483,E2 -11532.483} C_VEL
LIN {X 0,Y 390.143,Z 727.881,A -85,B 0,C 180,E1 -11535.677,E2 -11535.677} C_VEL
LIN {X 0,Y 390.108,Z 727.89,A -85,B 0,C 180,E1 -11538.922,E2 -11538.922} C_VEL
LIN {X 0,Y 390.041,Z 727.901,A -85,B 0,C 180,E1 -11542.234,E2 -11542.234} C_VEL
LIN {X 0,Y 390.122,Z 727.89,A -85,B 0,C 180,E1 -11545.743,E2 -11545.743} C_VEL
LIN {X 0,Y 390.061,Z 727.895,A -85,B 0,C 180,E1 -11549.109,E2 -11549.109} C_VEL
LIN {X 0,Y 390.046,Z 727.899,A -85,B 0,C 180,E1 -11552.721,E2 -11552.721} C_VEL
LIN {X 0,Y 390.059,Z 727.899,A -85,B 0,C 180,E1 -11555.825,E2 -11555.825} C_VEL
LIN {X 0,Y 390.073,Z 727.901,A -85,B 0,C 180,E1 -11559.218,E2 -11559.218} C_VEL
LIN {X 0,Y 390.045,Z 727.904,A -85,B 0,C 180,E1 -11562.374,E2 -11562.374} C_VEL
LIN {X 0,Y 390.052,Z 727.914,A -85,B 0,C 180,E1 -11564.84,E2 -11564.84} C_VEL
LIN {X 0,Y 391.804,Z 736.154,A -85,B 0,C 180,E1 -11568.418,E2 -11568.418} C_VEL
LIN {X 0,Y 393.203,Z 743.569,A -85,B 0,C 180,E1 -11571.275,E2 -11571.275} C_VEL
LIN {X 0,Y 393.757,Z 747.357,A -85,B 0,C 180,E1 -11572.637,E2 -11572.637} C_VEL
LIN {X 0,Y 393.148,Z 754.946,A -85,B 0,C 180,E1 -11575.107,E2 -11575.107} C_VEL
LIN {X 0,Y 392.293,Z 764.611,A -85,B 0,C 180,E1 -11578.096,E2 -11578.096} C_VEL
LIN {X 0,Y 391.319,Z 778.389,A -85,B 0,C 180,E1 -11582.163,E2 -11582.163} C_VEL
LIN {X 0,Y 390.643,Z 790.36,A -85,B 0,C 180,E1 -11585.557,E2 -11585.557} C_VEL
LIN {X 0,Y 390.025,Z 803.89,A -85,B 0,C 180,E1 -11589.284,E2 -11589.284} C_VEL
LIN {X 0,Y 389.842,Z 810.69,A -85,B 0,C 180,E1 -11591.09,E2 -11591.09} C_VEL
LIN {X 0,Y 391.581,Z 824.536,A -85,B 0,C 180,E1 -11591.635,E2 -11591.635} C_VEL
LIN {X 0,Y 392.436,Z 837.101,A -85,B 0,C 180,E1 -11592.275,E2 -11592.275} C_VEL
LIN {X 0,Y 392.902,Z 849.753,A -85,B 0,C 180,E1 -11593.102,E2 -11593.102} C_VEL
LIN {X 0,Y 393.123,Z 856.609,A -85,B 0,C 180,E1 -11593.646,E2 -11593.646} C_VEL
LIN {X 0,Y 392.096,Z 868.035,A -85,B 0,C 180,E1 -11594.67,E2 -11594.67} C_VEL
LIN {X 0,Y 391.257,Z 878.714,A -85,B 0,C 180,E1 -11595.857,E2 -11595.857} C_VEL
LIN {X 0,Y 390.803,Z 885.374,A -85,B 0,C 180,E1 -11596.745,E2 -11596.745} C_VEL
LIN {X 0,Y 390.145,Z 893.771,A -85,B 0,C 180,E1 -11598.044,E2 -11598.044} C_VEL
LIN {X 0,Y 389.594,Z 902.123,A -85,B 0,C 180,E1 -11599.607,E2 -11599.607} C_VEL
LIN {X 0,Y 389.36,Z 908.874,A -85,B 0,C 180,E1 -11601.174,E2 -11601.174} C_VEL
LIN {X 0,Y 389.243,Z 914.296,A -85,B 0,C 180,E1 -11602.739,E2 -11602.739} C_VEL
LIN {X 0,Y 389.271,Z 918.55,A -85,B 0,C 180,E1 -11604.301,E2 -11604.301} C_VEL
LIN {X 0,Y 389.427,Z 921.74,A -85,B 0,C 180,E1 -11605.86,E2 -11605.86} C_VEL
LIN {X 0,Y 389.384,Z 923.259,A -85,B 0,C 180,E1 -11606.896,E2 -11606.896} C_VEL
LIN {X 0,Y 389.4,Z 924.371,A -85,B 0,C 180,E1 -11607.931,E2 -11607.931} C_VEL
LIN {X 0,Y 389.419,Z 925.075,A -85,B 0,C 180,E1 -11608.966,E2 -11608.966} C_VEL
LIN {X 0,Y 389.439,Z 925.318,A -85,B 0,C 180,E1 -11610,E2 -11610} C_VEL
LIN {X 0,Y 389.413,Z 925.131,A -85,B 0,C 180,E1 -11611.034,E2 -11611.034} C_VEL
LIN {X 0,Y 389.386,Z 924.535,A -85,B 0,C 180,E1 -11612.069,E2 -11612.069} C_VEL
LIN {X 0,Y 389.374,Z 923.529,A -85,B 0,C 180,E1 -11613.104,E2 -11613.104} C_VEL
LIN {X 0,Y 389.45,Z 922.057,A -85,B 0,C 180,E1 -11614.139,E2 -11614.139} C_VEL
LIN {X 0,Y 389.24,Z 918.967,A -85,B 0,C 180,E1 -11615.699,E2 -11615.699} C_VEL
LIN {X 0,Y 389.258,Z 914.8,A -85,B 0,C 180,E1 -11617.261,E2 -11617.261} C_VEL
LIN {X 0,Y 389.375,Z 908.39,A -85,B 0,C 180,E1 -11619.087,E2 -11619.087} C_VEL
LIN {X 0,Y 389.668,Z 901.413,A -85,B 0,C 180,E1 -11620.653,E2 -11620.653} C_VEL
LIN {X 0,Y 390.16,Z 894.313,A -85,B 0,C 180,E1 -11621.955,E2 -11621.955} C_VEL
LIN {X 0,Y 390.886,Z 885.786,A -85,B 0,C 180,E1 -11623.252,E2 -11623.252} C_VEL
LIN {X 0,Y 391.422,Z 877.376,A -85,B 0,C 180,E1 -11624.317,E2 -11624.317} C_VEL
LIN {X 0,Y 392.204,Z 866.337,A -85,B 0,C 180,E1 -11625.459,E2 -11625.459} C_VEL
LIN {X 0,Y 393.125,Z 855.484,A -85,B 0,C 180,E1 -11626.354,E2 -11626.354} C_VEL
LIN {X 0,Y 392.361,Z 842.978,A -85,B 0,C 180,E1 -11627.208,E2 -11627.208} C_VEL
LIN {X 0,Y 391.327,Z 829.777,A -85,B 0,C 180,E1 -11627.886,E2 -11627.886} C_VEL
LIN {X 0,Y 389.837,Z 815.3,A -85,B 0,C 180,E1 -11628.411,E2 -11628.411} C_VEL
LIN {X 0,Y 390.343,Z 803.704,A -85,B 0,C 180,E1 -11631.66,E2 -11631.66} C_VEL
LIN {X 0,Y 391.156,Z 790.001,A -85,B 0,C 180,E1 -11635.545,E2 -11635.545} C_VEL
LIN {X 0,Y 391.98,Z 778.208,A -85,B 0,C 180,E1 -11638.953,E2 -11638.953} C_VEL
LIN {X 0,Y 393.073,Z 765.066,A -85,B 0,C 180,E1 -11642.824,E2 -11642.824} C_VEL
LIN {X 0,Y 394.115,Z 754.433,A -85,B 0,C 180,E1 -11646.048,E2 -11646.048} C_VEL
LIN {X 0,Y 394.395,Z 750.425,A -85,B 0,C 180,E1 -11647.292,E2 -11647.292} C_VEL
LIN {X 0,Y 393.421,Z 744.646,A -85,B 0,C 180,E1 -11649.207,E2 -11649.207} C_VEL
LIN {X 0,Y 391.522,Z 734.906,A -85,B 0,C 180,E1 -11652.611,E2 -11652.611} C_VEL
LIN {X 0,Y 390.047,Z 727.899,A -85,B 0,C 180,E1 -11655.255,E2 -11655.255} C_VEL
LIN {X 0,Y 390.033,Z 727.901,A -85,B 0,C 180,E1 -11658.187,E2 -11658.187} C_VEL
LIN {X 0,Y 390.091,Z 727.893,A -85,B 0,C 180,E1 -11660.908,E2 -11660.908} C_VEL
LIN {X 0,Y 390.087,Z 727.891,A -85,B 0,C 180,E1 -11664.793,E2 -11664.793} C_VEL
LIN {X 0,Y 390.034,Z 727.902,A -85,B 0,C 180,E1 -11667.875,E2 -11667.875} C_VEL
LIN {X 0,Y 390.06,Z 727.894,A -85,B 0,C 180,E1 -11670.891,E2 -11670.891} C_VEL
LIN {X 0,Y 390.121,Z 727.889,A -85,B 0,C 180,E1 -11674.257,E2 -11674.257} C_VEL
LIN {X 0,Y 390.04,Z 727.901,A -85,B 0,C 180,E1 -11677.766,E2 -11677.766} C_VEL
LIN {X 0,Y 390.107,Z 727.889,A -85,B 0,C 180,E1 -11681.078,E2 -11681.078} C_VEL
LIN {X 0,Y 390.141,Z 727.888,A -85,B 0,C 180,E1 -11684.323,E2 -11684.323} C_VEL
LIN {X 0,Y 390.173,Z 727.881,A -85,B 0,C 180,E1 -11687.517,E2 -11687.517} C_VEL
LIN {X 0,Y 390.207,Z 727.879,A -85,B 0,C 180,E1 -11690.671,E2 -11690.671} C_VEL
LIN {X 0,Y 390.327,Z 727.862,A -85,B 0,C 180,E1 -11693.798,E2 -11693.798} C_VEL
LIN {X 0,Y 390.415,Z 727.852,A -85,B 0,C 180,E1 -11697.937,E2 -11697.937} C_VEL
LIN {X 0,Y 390.546,Z 727.835,A -85,B 0,C 180,E1 -11700,E2 -11700} C_VEL
LIN {X 0,Y 390.304,Z 727.867,A -85,B 0,C 180,E1 -11703.097,E2 -11703.097} C_VEL
LIN {X 0,Y 390.277,Z 727.868,A -85,B 0,C 180,E1 -11706.513,E2 -11706.513} C_VEL
LIN {X 0,Y 390.195,Z 727.88,A -85,B 0,C 180,E1 -11709.329,E2 -11709.329} C_VEL
LIN {X 0,Y 390.173,Z 727.883,A -85,B 0,C 180,E1 -11712.483,E2 -11712.483} C_VEL
LIN {X 0,Y 390.141,Z 727.887,A -85,B 0,C 180,E1 -11715.677,E2 -11715.677} C_VEL
LIN {X 0,Y 390.105,Z 727.894,A -85,B 0,C 180,E1 -11718.922,E2 -11718.922} C_VEL
LIN {X 0,Y 390.037,Z 727.898,A -85,B 0,C 180,E1 -11722.235,E2 -11722.235} C_VEL
LIN {X 0,Y 390.051,Z 727.899,A -85,B 0,C 180,E1 -11725.722,E2 -11725.722} C_VEL
LIN {X 0,Y 390.035,Z 727.902,A -85,B 0,C 180,E1 -11729.112,E2 -11729.112} C_VEL
LIN {X 0,Y 390.043,Z 727.898,A -85,B 0,C 180,E1 -11732.722,E2 -11732.722} C_VEL
LIN {X 0,Y 390.044,Z 727.9,A -85,B 0,C 180,E1 -11735.823,E2 -11735.823} C_VEL
LIN {X 0,Y 390.038,Z 727.9,A -85,B 0,C 180,E1 -11739.212,E2 -11739.212} C_VEL
LIN {X 0,Y 390.031,Z 727.901,A -85,B 0,C 180,E1 -11742.372,E2 -11742.372} C_VEL
LIN {X 0,Y 390.041,Z 727.899,A -85,B 0,C 180,E1 -11745.354,E2 -11745.354} C_VEL
LIN {X 0,Y 390.016,Z 727.904,A -85,B 0,C 180,E1 -11748.185,E2 -11748.185} C_VEL
LIN {X 0,Y 390.058,Z 727.896,A -85,B 0,C 180,E1 -11750.904,E2 -11750.904} C_VEL
LIN {X 0,Y 390.069,Z 727.896,A -85,B 0,C 180,E1 -11754.791,E2 -11754.791} C_VEL
LIN {X 0,Y 390.019,Z 727.904,A -85,B 0,C 180,E1 -11758.495,E2 -11758.495} C_VEL
LIN {X 0,Y 390.017,Z 727.903,A -85,B 0,C 180,E1 -11762.003,E2 -11762.003} C_VEL
LIN {X 0,Y 390.043,Z 727.898,A -85,B 0,C 180,E1 -11765.517,E2 -11765.517} C_VEL
LIN {X 0,Y 390.058,Z 727.9,A -85,B 0,C 180,E1 -11768.878,E2 -11768.878} C_VEL
LIN {X 0,Y 390.114,Z 727.891,A -85,B 0,C 180,E1 -11772.166,E2 -11772.166} C_VEL
LIN {X 0,Y 390.144,Z 727.886,A -85,B 0,C 180,E1 -11775.393,E2 -11775.393} C_VEL
LIN {X 0,Y 390.138,Z 727.888,A -85,B 0,C 180,E1 -11778.571,E2 -11778.571} C_VEL
LIN {X 0,Y 390.259,Z 727.871,A -85,B 0,C 180,E1 -11782.086,E2 -11782.086} C_VEL
LIN {X 0,Y 390.201,Z 727.88,A -85,B 0,C 180,E1 -11784.833,E2 -11784.833} C_VEL
LIN {X 0,Y 390.409,Z 727.852,A -85,B 0,C 180,E1 -11787.937,E2 -11787.937} C_VEL
LIN {X 0,Y 390.41,Z 727.852,A -85,B 0,C 180,E1 -11792.063,E2 -11792.063} C_VEL
LIN {X 0,Y 390.286,Z 727.867,A -85,B 0,C 180,E1 -11796.203,E2 -11796.203} C_VEL
LIN {X 0,Y 390.195,Z 727.881,A -85,B 0,C 180,E1 -11799.329,E2 -11799.329} C_VEL
LIN {X 0,Y 390.174,Z 727.88,A -85,B 0,C 180,E1 -11802.483,E2 -11802.483} C_VEL
LIN {X 0,Y 390.143,Z 727.89,A -85,B 0,C 180,E1 -11805.677,E2 -11805.677} C_VEL
LIN {X 0,Y 390.108,Z 727.889,A -85,B 0,C 180,E1 -11808.922,E2 -11808.922} C_VEL
LIN {X 0,Y 390.04,Z 727.899,A -85,B 0,C 180,E1 -11812.234,E2 -11812.234} C_VEL
LIN {X 0,Y 390.053,Z 727.899,A -85,B 0,C 180,E1 -11815.722,E2 -11815.722} C_VEL
LIN {X 0,Y 390.036,Z 727.897,A -85,B 0,C 180,E1 -11819.112,E2 -11819.112} C_VEL
LIN {X 0,Y 390.014,Z 727.9,A -85,B 0,C 180,E1 -11820.792,E2 -11820.792} C_VEL
LIN {X 0,Y 389.341,Z 727.987,A -85,B 0,C 180,E1 -11821.654,E2 -11821.654} C_VEL
LIN {X 0,Y 386.494,Z 728.338,A -85,B 0,C 180,E1 -11823.055,E2 -11823.055} C_VEL
LIN {X 0,Y 384.097,Z 728.643,A -85,B 0,C 180,E1 -11824.188,E2 -11824.188} C_VEL
LIN {X 0,Y 383.078,Z 728.764,A -85,B 0,C 180,E1 -11825.064,E2 -11825.064} C_VEL
LIN {X 0,Y 383.001,Z 728.773,A -85,B 0,C 180,E1 -11825.361,E2 -11825.361} C_VEL
LIN {X 0,Y 383.005,Z 728.775,A -85,B 0,C 180,E1 -11828.601,E2 -11828.601} C_VEL
LIN {X 0,Y 382.987,Z 728.775,A -85,B 0,C 180,E1 -11831.347,E2 -11831.347} C_VEL
LIN {X 0,Y 383.053,Z 728.925,A -85,B 0,C 180,E1 -11834.624,E2 -11834.624} C_VEL
LIN {X 0,Y 386.37,Z 740.441,A -85,B 0,C 180,E1 -11835.523,E2 -11835.523} C_VEL
LIN {X 0,Y 387.758,Z 746.034,A -85,B 0,C 180,E1 -11836.027,E2 -11836.027} C_VEL
LIN {X 0,Y 387.104,Z 757.672,A -85,B 0,C 180,E1 -11837.091,E2 -11837.091} C_VEL
LIN {X 0,Y 386.412,Z 768.437,A -85,B 0,C 180,E1 -11838.317,E2 -11838.317} C_VEL
LIN {X 0,Y 385.803,Z 777.271,A -85,B 0,C 180,E1 -11839.556,E2 -11839.556} C_VEL
LIN {X 0,Y 385.102,Z 785.628,A -85,B 0,C 180,E1 -11840.978,E2 -11840.978} C_VEL
LIN {X 0,Y 384.512,Z 793.251,A -85,B 0,C 180,E1 -11842.574,E2 -11842.574} C_VEL
LIN {X 0,Y 384.033,Z 799.319,A -85,B 0,C 180,E1 -11844.153,E2 -11844.153} C_VEL
LIN {X 0,Y 383.567,Z 805.018,A -85,B 0,C 180,E1 -11846.083,E2 -11846.083} C_VEL
LIN {X 0,Y 383.364,Z 808.883,A -85,B 0,C 180,E1 -11847.883,E2 -11847.883} C_VEL
LIN {X 0,Y 383.177,Z 811.333,A -85,B 0,C 180,E1 -11849.548,E2 -11849.548} C_VEL
LIN {X 0,Y 383.111,Z 812.975,A -85,B 0,C 180,E1 -11851.708,E2 -11851.708} C_VEL
LIN {X 0,Y 383.154,Z 813.157,A -85,B 0,C 180,E1 -11852.705,E2 -11852.705} C_VEL
LIN {X 0,Y 383.3,Z 812.905,A -85,B 0,C 180,E1 -11853.955,E2 -11853.955} C_VEL
LIN {X 0,Y 383.466,Z 812.16,A -85,B 0,C 180,E1 -11855.068,E2 -11855.068} C_VEL
LIN {X 0,Y 383.671,Z 810.811,A -85,B 0,C 180,E1 -11856.333,E2 -11856.333} C_VEL
LIN {X 0,Y 384.08,Z 808.134,A -85,B 0,C 180,E1 -11857.968,E2 -11857.968} C_VEL
LIN {X 0,Y 384.626,Z 804.132,A -85,B 0,C 180,E1 -11859.685,E2 -11859.685} C_VEL
LIN {X 0,Y 385.347,Z 798.356,A -85,B 0,C 180,E1 -11861.512,E2 -11861.512} C_VEL
LIN {X 0,Y 386.074,Z 792.063,A -85,B 0,C 180,E1 -11863.066,E2 -11863.066} C_VEL
LIN {X 0,Y 386.945,Z 784.553,A -85,B 0,C 180,E1 -11864.554,E2 -11864.554} C_VEL
LIN {X 0,Y 387.737,Z 776.608,A -85,B 0,C 180,E1 -11865.836,E2 -11865.836} C_VEL
LIN {X 0,Y 388.682,Z 765.936,A -85,B 0,C 180,E1 -11867.229,E2 -11867.229} C_VEL
LIN {X 0,Y 389.45,Z 755.017,A -85,B 0,C 180,E1 -11868.371,E2 -11868.371} C_VEL
LIN {X 0,Y 389.834,Z 749.454,A -85,B 0,C 180,E1 -11868.851,E2 -11868.851} C_VEL
LIN {X 0,Y 387.008,Z 739.662,A -85,B 0,C 180,E1 -11869.802,E2 -11869.802} C_VEL
LIN {X 0,Y 383.173,Z 728.756,A -85,B 0,C 180,E1 -11870.731,E2 -11870.731} C_VEL
LIN {X 0,Y 383.253,Z 728.746,A -85,B 0,C 180,E1 -11873.683,E2 -11873.683} C_VEL
LIN {X 0,Y 383.387,Z 728.732,A -85,B 0,C 180,E1 -11877.899,E2 -11877.899} C_VEL
LIN {X 0,Y 383.517,Z 728.714,A -85,B 0,C 180,E1 -11880,E2 -11880} C_VEL
LIN {X 0,Y 383.243,Z 728.74,A -85,B 0,C 180,E1 -11883.154,E2 -11883.154} C_VEL
LIN {X 0,Y 383.28,Z 728.739,A -85,B 0,C 180,E1 -11886.316,E2 -11886.316} C_VEL
LIN {X 0,Y 383.224,Z 728.743,A -85,B 0,C 180,E1 -11888.436,E2 -11888.436} C_VEL
LIN {X 0,Y 383.101,Z 728.761,A -85,B 0,C 180,E1 -11891.642,E2 -11891.642} C_VEL
LIN {X 0,Y 383.114,Z 728.755,A -85,B 0,C 180,E1 -11894.882,E2 -11894.882} C_VEL
LIN {X 0,Y 383.066,Z 728.765,A -85,B 0,C 180,E1 -11898.173,E2 -11898.173} C_VEL
LIN {X 0,Y 382.996,Z 728.771,A -85,B 0,C 180,E1 -11901.531,E2 -11901.531} C_VEL
LIN {X 0,Y 383.054,Z 728.77,A -85,B 0,C 180,E1 -11904.96,E2 -11904.96} C_VEL
LIN {X 0,Y 383.033,Z 728.773,A -85,B 0,C 180,E1 -11908.27,E2 -11908.27} C_VEL
LIN {X 0,Y 383.013,Z 728.777,A -85,B 0,C 180,E1 -11912.149,E2 -11912.149} C_VEL
LIN {X 0,Y 383.021,Z 728.776,A -85,B 0,C 180,E1 -11914.668,E2 -11914.668} C_VEL
LIN {X 0,Y 383.003,Z 728.781,A -85,B 0,C 180,E1 -11917.904,E2 -11917.904} C_VEL
LIN {X 0,Y 382.987,Z 728.783,A -85,B 0,C 180,E1 -11921.347,E2 -11921.347} C_VEL
LIN {X 0,Y 383.008,Z 728.852,A -85,B 0,C 180,E1 -11924.305,E2 -11924.305} C_VEL
LIN {X 0,Y 384.681,Z 736.772,A -85,B 0,C 180,E1 -11927.87,E2 -11927.87} C_VEL
LIN {X 0,Y 385.918,Z 743.027,A -85,B 0,C 180,E1 -11930.402,E2 -11930.402} C_VEL
LIN {X 0,Y 386.835,Z 748.685,A -85,B 0,C 180,E1 -11932.51,E2 -11932.51} C_VEL
LIN {X 0,Y 386.197,Z 756.078,A -85,B 0,C 180,E1 -11934.976,E2 -11934.976} C_VEL
LIN {X 0,Y 385.284,Z 765.835,A -85,B 0,C 180,E1 -11938.062,E2 -11938.062} C_VEL
LIN {X 0,Y 384.248,Z 779.538,A -85,B 0,C 180,E1 -11942.199,E2 -11942.199} C_VEL
LIN {X 0,Y 383.551,Z 791.458,A -85,B 0,C 180,E1 -11945.652,E2 -11945.652} C_VEL
LIN {X 0,Y 382.994,Z 803.294,A -85,B 0,C 180,E1 -11948.996,E2 -11948.996} C_VEL
LIN {X 0,Y 382.767,Z 809.184,A -85,B 0,C 180,E1 -11950.631,E2 -11950.631} C_VEL
LIN {X 0,Y 384.777,Z 824.255,A -85,B 0,C 180,E1 -11951.273,E2 -11951.273} C_VEL
LIN {X 0,Y 385.581,Z 836.854,A -85,B 0,C 180,E1 -11951.949,E2 -11951.949} C_VEL
LIN {X 0,Y 385.906,Z 849.134,A -85,B 0,C 180,E1 -11952.786,E2 -11952.786} C_VEL
LIN {X 0,Y 386.255,Z 855.944,A -85,B 0,C 180,E1 -11953.347,E2 -11953.347} C_VEL
LIN {X 0,Y 385.228,Z 867.289,A -85,B 0,C 180,E1 -11954.389,E2 -11954.389} C_VEL
LIN {X 0,Y 384.305,Z 877.941,A -85,B 0,C 180,E1 -11955.604,E2 -11955.604} C_VEL
LIN {X 0,Y 383.778,Z 884.507,A -85,B 0,C 180,E1 -11956.497,E2 -11956.497} C_VEL
LIN {X 0,Y 383.122,Z 892.872,A -85,B 0,C 180,E1 -11957.821,E2 -11957.821} C_VEL
LIN {X 0,Y 382.544,Z 901.167,A -85,B 0,C 180,E1 -11959.413,E2 -11959.413} C_VEL
LIN {X 0,Y 382.294,Z 907.881,A -85,B 0,C 180,E1 -11961.01,E2 -11961.01} C_VEL
LIN {X 0,Y 382.165,Z 913.29,A -85,B 0,C 180,E1 -11962.604,E2 -11962.604} C_VEL
LIN {X 0,Y 382.212,Z 917.541,A -85,B 0,C 180,E1 -11964.195,E2 -11964.195} C_VEL
LIN {X 0,Y 382.361,Z 920.725,A -85,B 0,C 180,E1 -11965.784,E2 -11965.784} C_VEL
LIN {X 0,Y 382.341,Z 922.247,A -85,B 0,C 180,E1 -11966.839,E2 -11966.839} C_VEL
LIN {X 0,Y 382.361,Z 923.36,A -85,B 0,C 180,E1 -11967.893,E2 -11967.893} C_VEL
LIN {X 0,Y 382.387,Z 924.057,A -85,B 0,C 180,E1 -11968.947,E2 -11968.947} C_VEL
LIN {X 0,Y 382.414,Z 924.289,A -85,B 0,C 180,E1 -11970,E2 -11970} C_VEL
LIN {X 0,Y 382.384,Z 924.095,A -85,B 0,C 180,E1 -11971.053,E2 -11971.053} C_VEL
LIN {X 0,Y 382.352,Z 923.495,A -85,B 0,C 180,E1 -11972.107,E2 -11972.107} C_VEL
LIN {X 0,Y 382.34,Z 922.476,A -85,B 0,C 180,E1 -11973.161,E2 -11973.161} C_VEL
LIN {X 0,Y 382.393,Z 920.984,A -85,B 0,C 180,E1 -11974.216,E2 -11974.216} C_VEL
LIN {X 0,Y 382.188,Z 917.874,A -85,B 0,C 180,E1 -11975.805,E2 -11975.805} C_VEL
LIN {X 0,Y 382.219,Z 913.683,A -85,B 0,C 180,E1 -11977.395,E2 -11977.395} C_VEL
LIN {X 0,Y 382.331,Z 907.245,A -85,B 0,C 180,E1 -11979.256,E2 -11979.256} C_VEL
LIN {X 0,Y 382.644,Z 900.235,A -85,B 0,C 180,E1 -11980.851,E2 -11980.851} C_VEL
LIN {X 0,Y 383.216,Z 891.466,A -85,B 0,C 180,E1 -11982.444,E2 -11982.444} C_VEL
LIN {X 0,Y 383.865,Z 884.502,A -85,B 0,C 180,E1 -11983.499,E2 -11983.499} C_VEL
LIN {X 0,Y 384.52,Z 875.078,A -85,B 0,C 180,E1 -11984.692,E2 -11984.692} C_VEL
LIN {X 0,Y 385.474,Z 863.546,A -85,B 0,C 180,E1 -11985.872,E2 -11985.872} C_VEL
LIN {X 0,Y 386.112,Z 853.979,A -85,B 0,C 180,E1 -11986.659,E2 -11986.659} C_VEL
LIN {X 0,Y 385.313,Z 842.19,A -85,B 0,C 180,E1 -11987.481,E2 -11987.481} C_VEL
LIN {X 0,Y 384.282,Z 828.872,A -85,B 0,C 180,E1 -11988.183,E2 -11988.183} C_VEL
LIN {X 0,Y 382.771,Z 814.289,A -85,B 0,C 180,E1 -11988.742,E2 -11988.742} C_VEL
LIN {X 0,Y 383.327,Z 802.67,A -85,B 0,C 180,E1 -11992.077,E2 -11992.077} C_VEL
LIN {X 0,Y 384.049,Z 790.976,A -85,B 0,C 180,E1 -11995.47,E2 -11995.47} C_VEL
LIN {X 0,Y 384.971,Z 778.633,A -85,B 0,C 180,E1 -11999.1,E2 -11999.1} C_VEL
LIN {X 0,Y 386.154,Z 765.21,A -85,B 0,C 180,E1 -12003.154,E2 -12003.154} C_VEL
LIN {X 0,Y 387.13,Z 755.467,A -85,B 0,C 180,E1 -12006.158,E2 -12006.158} C_VEL
LIN {X 0,Y 387.409,Z 751.243,A -85,B 0,C 180,E1 -12007.501,E2 -12007.501} C_VEL
LIN {X 0,Y 385.998,Z 743.595,A -85,B 0,C 180,E1 -12010.119,E2 -12010.119} C_VEL
LIN {X 0,Y 384.42,Z 735.557,A -85,B 0,C 180,E1 -12013.006,E2 -12013.006} C_VEL
LIN {X 0,Y 383.023,Z 728.775,A -85,B 0,C 180,E1 -12015.602,E2 -12015.602} C_VEL
LIN {X 0,Y 382.989,Z 728.779,A -85,B 0,C 180,E1 -12018.796,E2 -12018.796} C_VEL
LIN {X 0,Y 383.001,Z 728.775,A -85,B 0,C 180,E1 -12022.096,E2 -12022.096} C_VEL
LIN {X 0,Y 383.02,Z 728.774,A -85,B 0,C 180,E1 -12025.332,E2 -12025.332} C_VEL
LIN {X 0,Y 382.984,Z 728.776,A -85,B 0,C 180,E1 -12029.082,E2 -12029.082} C_VEL
LIN {X 0,Y 383.058,Z 728.767,A -85,B 0,C 180,E1 -12032.698,E2 -12032.698} C_VEL
LIN {X 0,Y 383.052,Z 728.767,A -85,B 0,C 180,E1 -12035.04,E2 -12035.04} C_VEL
LIN {X 0,Y 382.994,Z 728.777,A -85,B 0,C 180,E1 -12038.469,E2 -12038.469} C_VEL
LIN {X 0,Y 383.091,Z 728.766,A -85,B 0,C 180,E1 -12041.828,E2 -12041.828} C_VEL
LIN {X 0,Y 383.112,Z 728.76,A -85,B 0,C 180,E1 -12045.118,E2 -12045.118} C_VEL
LIN {X 0,Y 383.099,Z 728.766,A -85,B 0,C 180,E1 -12048.358,E2 -12048.358} C_VEL
LIN {X 0,Y 383.266,Z 728.743,A -85,B 0,C 180,E1 -12051.976,E2 -12051.976} C_VEL
LIN {X 0,Y 383.196,Z 728.753,A -85,B 0,C 180,E1 -12054.739,E2 -12054.739} C_VEL
LIN {X 0,Y 383.381,Z 728.727,A -85,B 0,C 180,E1 -12057.899,E2 -12057.899} C_VEL
LIN {X 0,Y 383.516,Z 728.711,A -85,B 0,C 180,E1 -12060,E2 -12060} C_VEL
LIN {X 0,Y 383.24,Z 728.747,A -85,B 0,C 180,E1 -12063.154,E2 -12063.154} C_VEL
LIN {X 0,Y 383.24,Z 728.745,A -85,B 0,C 180,E1 -12066.501,E2 -12066.501} C_VEL
LIN {X 0,Y 383.145,Z 728.758,A -85,B 0,C 180,E1 -12069.502,E2 -12069.502} C_VEL
LIN {X 0,Y 383.128,Z 728.761,A -85,B 0,C 180,E1 -12073.536,E2 -12073.536} C_VEL
LIN {X 0,Y 383.096,Z 728.766,A -85,B 0,C 180,E1 -12077.069,E2 -12077.069} C_VEL
LIN {X 0,Y 383.031,Z 728.772,A -85,B 0,C 180,E1 -12080.647,E2 -12080.647} C_VEL
LIN {X 0,Y 383.011,Z 728.776,A -85,B 0,C 180,E1 -12083.809,E2 -12083.809} C_VEL
LIN {X 0,Y 382.993,Z 728.779,A -85,B 0,C 180,E1 -12087.307,E2 -12087.307} C_VEL
LIN {X 0,Y 382.984,Z 728.778,A -85,B 0,C 180,E1 -12090.919,E2 -12090.919} C_VEL
LIN {X 0,Y 383.013,Z 728.773,A -85,B 0,C 180,E1 -12094.669,E2 -12094.669} C_VEL
LIN {X 0,Y 382.994,Z 728.778,A -85,B 0,C 180,E1 -12097.902,E2 -12097.902} C_VEL
LIN {X 0,Y 382.962,Z 728.782,A -85,B 0,C 180,E1 -12101.351,E2 -12101.351} C_VEL
LIN {X 0,Y 382.99,Z 728.779,A -85,B 0,C 180,E1 -12104.302,E2 -12104.302} C_VEL
LIN {X 0,Y 382.998,Z 728.776,A -85,B 0,C 180,E1 -12107.238,E2 -12107.238} C_VEL
LIN {X 0,Y 382.986,Z 728.78,A -85,B 0,C 180,E1 -12110.419,E2 -12110.419} C_VEL
LIN {X 0,Y 383.014,Z 728.776,A -85,B 0,C 180,E1 -12114.043,E2 -12114.043} C_VEL
LIN {X 0,Y 382.983,Z 728.778,A -85,B 0,C 180,E1 -12117.58,E2 -12117.58} C_VEL
LIN {X 0,Y 382.976,Z 728.781,A -85,B 0,C 180,E1 -12120.299,E2 -12120.299} C_VEL
LIN {X 0,Y 383.004,Z 728.777,A -85,B 0,C 180,E1 -12124.045,E2 -12124.045} C_VEL
LIN {X 0,Y 382.991,Z 728.776,A -85,B 0,C 180,E1 -12127.334,E2 -12127.334} C_VEL
LIN {X 0,Y 383.061,Z 728.771,A -85,B 0,C 180,E1 -12130.716,E2 -12130.716} C_VEL
LIN {X 0,Y 383.081,Z 728.765,A -85,B 0,C 180,E1 -12134.027,E2 -12134.027} C_VEL
LIN {X 0,Y 383.136,Z 728.76,A -85,B 0,C 180,E1 -12137.284,E2 -12137.284} C_VEL
LIN {X 0,Y 383.138,Z 728.76,A -85,B 0,C 180,E1 -12140.498,E2 -12140.498} C_VEL
LIN {X 0,Y 383.236,Z 728.746,A -85,B 0,C 180,E1 -12143.683,E2 -12143.683} C_VEL
LIN {X 0,Y 383.375,Z 728.728,A -85,B 0,C 180,E1 -12147.899,E2 -12147.899} C_VEL
LIN {X 0,Y 383.376,Z 728.728,A -85,B 0,C 180,E1 -12152.101,E2 -12152.101} C_VEL
LIN {X 0,Y 383.243,Z 728.744,A -85,B 0,C 180,E1 -12156.317,E2 -12156.317} C_VEL
LIN {X 0,Y 383.146,Z 728.761,A -85,B 0,C 180,E1 -12159.502,E2 -12159.502} C_VEL
LIN {X 0,Y 383.129,Z 728.762,A -85,B 0,C 180,E1 -12163.536,E2 -12163.536} C_VEL
LIN {X 0,Y 383.098,Z 728.765,A -85,B 0,C 180,E1 -12167.455,E2 -12167.455} C_VEL
LIN {X 0,Y 383.032,Z 728.77,A -85,B 0,C 180,E1 -12170.647,E2 -12170.647} C_VEL
LIN {X 0,Y 383.017,Z 728.777,A -85,B 0,C 180,E1 -12173.809,E2 -12173.809} C_VEL
LIN {X 0,Y 382.996,Z 728.775,A -85,B 0,C 180,E1 -12177.307,E2 -12177.307} C_VEL
LIN {X 0,Y 382.985,Z 728.775,A -85,B 0,C 180,E1 -12180.919,E2 -12180.919} C_VEL
LIN {X 0,Y 383.021,Z 728.772,A -85,B 0,C 180,E1 -12184.668,E2 -12184.668} C_VEL
LIN {X 0,Y 383.001,Z 728.773,A -85,B 0,C 180,E1 -12185.361,E2 -12185.361} C_VEL
LIN {X 0,Y 382.363,Z 728.859,A -85,B 0,C 180,E1 -12186.238,E2 -12186.238} C_VEL
LIN {X 0,Y 379.568,Z 729.209,A -85,B 0,C 180,E1 -12187.667,E2 -12187.667} C_VEL
LIN {X 0,Y 377.165,Z 729.509,A -85,B 0,C 180,E1 -12188.821,E2 -12188.821} C_VEL
LIN {X 0,Y 376.094,Z 729.638,A -85,B 0,C 180,E1 -12189.713,E2 -12189.713} C_VEL
LIN {X 0,Y 375.986,Z 729.65,A -85,B 0,C 180,E1 -12190.015,E2 -12190.015} C_VEL
LIN {X 0,Y 375.936,Z 729.654,A -85,B 0,C 180,E1 -12193.766,E2 -12193.766} C_VEL
LIN {X 0,Y 376,Z 729.794,A -85,B 0,C 180,E1 -12194.344,E2 -12194.344} C_VEL
LIN {X 0,Y 379.314,Z 741.169,A -85,B 0,C 180,E1 -12195.245,E2 -12195.245} C_VEL
LIN {X 0,Y 380.902,Z 747.851,A -85,B 0,C 180,E1 -12195.861,E2 -12195.861} C_VEL
LIN {X 0,Y 380.163,Z 759.836,A -85,B 0,C 180,E1 -12196.994,E2 -12196.994} C_VEL
LIN {X 0,Y 379.503,Z 769.942,A -85,B 0,C 180,E1 -12198.188,E2 -12198.188} C_VEL
LIN {X 0,Y 378.81,Z 779.152,A -85,B 0,C 180,E1 -12199.523,E2 -12199.523} C_VEL
LIN {X 0,Y 378.046,Z 788.225,A -85,B 0,C 180,E1 -12201.136,E2 -12201.136} C_VEL
LIN {X 0,Y 377.451,Z 795.39,A -85,B 0,C 180,E1 -12202.721,E2 -12202.721} C_VEL
LIN {X 0,Y 376.963,Z 801.325,A -85,B 0,C 180,E1 -12204.365,E2 -12204.365} C_VEL
LIN {X 0,Y 376.577,Z 805.867,A -85,B 0,C 180,E1 -12205.952,E2 -12205.952} C_VEL
LIN {X 0,Y 376.34,Z 809.893,A -85,B 0,C 180,E1 -12207.844,E2 -12207.844} C_VEL
LIN {X 0,Y 376.14,Z 812.56,A -85,B 0,C 180,E1 -12209.703,E2 -12209.703} C_VEL
LIN {X 0,Y 376.11,Z 813.917,A -85,B 0,C 180,E1 -12211.432,E2 -12211.432} C_VEL
LIN {X 0,Y 376.239,Z 814.081,A -85,B 0,C 180,E1 -12213.718,E2 -12213.718} C_VEL
LIN {X 0,Y 376.576,Z 812.726,A -85,B 0,C 180,E1 -12215.758,E2 -12215.758} C_VEL
LIN {X 0,Y 376.822,Z 811.22,A -85,B 0,C 180,E1 -12216.942,E2 -12216.942} C_VEL
LIN {X 0,Y 377.292,Z 808.15,A -85,B 0,C 180,E1 -12218.651,E2 -12218.651} C_VEL
LIN {X 0,Y 377.887,Z 803.667,A -85,B 0,C 180,E1 -12220.441,E2 -12220.441} C_VEL
LIN {X 0,Y 378.704,Z 797.893,A -85,B 0,C 180,E1 -12222.169,E2 -12222.169} C_VEL
LIN {X 0,Y 379.636,Z 790.569,A -85,B 0,C 180,E1 -12223.878,E2 -12223.878} C_VEL
LIN {X 0,Y 380.502,Z 783.073,A -85,B 0,C 180,E1 -12225.287,E2 -12225.287} C_VEL
LIN {X 0,Y 381.442,Z 773.959,A -85,B 0,C 180,E1 -12226.684,E2 -12226.684} C_VEL
LIN {X 0,Y 382.371,Z 763.176,A -85,B 0,C 180,E1 -12228.003,E2 -12228.003} C_VEL
LIN {X 0,Y 383.167,Z 752.242,A -85,B 0,C 180,E1 -12229.072,E2 -12229.072} C_VEL
LIN {X 0,Y 382.633,Z 748.716,A -85,B 0,C 180,E1 -12229.416,E2 -12229.416} C_VEL
LIN {X 0,Y 378.964,Z 737.412,A -85,B 0,C 180,E1 -12230.527,E2 -12230.527} C_VEL
LIN {X 0,Y 376.181,Z 730.035,A -85,B 0,C 180,E1 -12231.167,E2 -12231.167} C_VEL
LIN {X 0,Y 376.127,Z 729.635,A -85,B 0,C 180,E1 -12231.2,E2 -12231.2} C_VEL
LIN {X 0,Y 376.21,Z 729.625,A -85,B 0,C 180,E1 -12233.564,E2 -12233.564} C_VEL
LIN {X 0,Y 376.353,Z 729.607,A -85,B 0,C 180,E1 -12237.859,E2 -12237.859} C_VEL
LIN {X 0,Y 376.487,Z 729.59,A -85,B 0,C 180,E1 -12240,E2 -12240} C_VEL
LIN {X 0,Y 376.353,Z 729.602,A -85,B 0,C 180,E1 -12242.14,E2 -12242.14} C_VEL
LIN {X 0,Y 376.238,Z 729.616,A -85,B 0,C 180,E1 -12246.435,E2 -12246.435} C_VEL
LIN {X 0,Y 376.119,Z 729.628,A -85,B 0,C 180,E1 -12249.681,E2 -12249.681} C_VEL
LIN {X 0,Y 376.093,Z 729.637,A -85,B 0,C 180,E1 -12253.658,E2 -12253.658} C_VEL
LIN {X 0,Y 376.047,Z 729.641,A -85,B 0,C 180,E1 -12257.607,E2 -12257.607} C_VEL
LIN {X 0,Y 375.981,Z 729.645,A -85,B 0,C 180,E1 -12260.832,E2 -12260.832} C_VEL
LIN {X 0,Y 375.991,Z 729.647,A -85,B 0,C 180,E1 -12264.282,E2 -12264.282} C_VEL
LIN {X 0,Y 376.023,Z 729.643,A -85,B 0,C 180,E1 -12266.652,E2 -12266.652} C_VEL
LIN {X 0,Y 375.967,Z 729.655,A -85,B 0,C 180,E1 -12270.312,E2 -12270.312} C_VEL
LIN {X 0,Y 375.965,Z 729.655,A -85,B 0,C 180,E1 -12274.111,E2 -12274.111} C_VEL
LIN {X 0,Y 375.956,Z 729.657,A -85,B 0,C 180,E1 -12276.741,E2 -12276.741} C_VEL
LIN {X 0,Y 375.991,Z 729.655,A -85,B 0,C 180,E1 -12279.971,E2 -12279.971} C_VEL
LIN {X 0,Y 375.977,Z 729.852,A -85,B 0,C 180,E1 -12283.759,E2 -12283.759} C_VEL
LIN {X 0,Y 377.579,Z 737.319,A -85,B 0,C 180,E1 -12287.278,E2 -12287.278} C_VEL
LIN {X 0,Y 379,Z 744.439,A -85,B 0,C 180,E1 -12290.253,E2 -12290.253} C_VEL
LIN {X 0,Y 379.887,Z 749.958,A -85,B 0,C 180,E1 -12292.373,E2 -12292.373} C_VEL
LIN {X 0,Y 379.466,Z 755.26,A -85,B 0,C 180,E1 -12294.2,E2 -12294.2} C_VEL
LIN {X 0,Y 378.496,Z 765.091,A -85,B 0,C 180,E1 -12297.42,E2 -12297.42} C_VEL
LIN {X 0,Y 377.309,Z 778.737,A -85,B 0,C 180,E1 -12301.653,E2 -12301.653} C_VEL
LIN {X 0,Y 376.556,Z 790.535,A -85,B 0,C 180,E1 -12305.169,E2 -12305.169} C_VEL
LIN {X 0,Y 375.982,Z 802.478,A -85,B 0,C 180,E1 -12308.623,E2 -12308.623} C_VEL
LIN {X 0,Y 375.736,Z 807.934,A -85,B 0,C 180,E1 -12310.183,E2 -12310.183} C_VEL
LIN {X 0,Y 377.858,Z 822.991,A -85,B 0,C 180,E1 -12310.846,E2 -12310.846} C_VEL
LIN {X 0,Y 378.729,Z 835.449,A -85,B 0,C 180,E1 -12311.534,E2 -12311.534} C_VEL
LIN {X 0,Y 378.962,Z 846.992,A -85,B 0,C 180,E1 -12312.325,E2 -12312.325} C_VEL
LIN {X 0,Y 379.302,Z 856.959,A -85,B 0,C 180,E1 -12313.171,E2 -12313.171} C_VEL
LIN {X 0,Y 378.217,Z 867.813,A -85,B 0,C 180,E1 -12314.231,E2 -12314.231} C_VEL
LIN {X 0,Y 377.253,Z 878.267,A -85,B 0,C 180,E1 -12315.489,E2 -12315.489} C_VEL
LIN {X 0,Y 376.58,Z 887.161,A -85,B 0,C 180,E1 -12316.784,E2 -12316.784} C_VEL
LIN {X 0,Y 375.828,Z 896.339,A -85,B 0,C 180,E1 -12318.403,E2 -12318.403} C_VEL
LIN {X 0,Y 375.4,Z 903.759,A -85,B 0,C 180,E1 -12320.027,E2 -12320.027} C_VEL
LIN {X 0,Y 375.139,Z 910.65,A -85,B 0,C 180,E1 -12321.923,E2 -12321.923} C_VEL
LIN {X 0,Y 375.151,Z 915.26,A -85,B 0,C 180,E1 -12323.546,E2 -12323.546} C_VEL
LIN {X 0,Y 375.17,Z 917.735,A -85,B 0,C 180,E1 -12324.625,E2 -12324.625} C_VEL
LIN {X 0,Y 375.295,Z 919.715,A -85,B 0,C 180,E1 -12325.704,E2 -12325.704} C_VEL
LIN {X 0,Y 375.299,Z 921.239,A -85,B 0,C 180,E1 -12326.779,E2 -12326.779} C_VEL
LIN {X 0,Y 375.321,Z 922.349,A -85,B 0,C 180,E1 -12327.854,E2 -12327.854} C_VEL
LIN {X 0,Y 375.356,Z 923.036,A -85,B 0,C 180,E1 -12328.927,E2 -12328.927} C_VEL
LIN {X 0,Y 375.388,Z 923.261,A -85,B 0,C 180,E1 -12330,E2 -12330} C_VEL
LIN {X 0,Y 375.355,Z 923.063,A -85,B 0,C 180,E1 -12331.073,E2 -12331.073} C_VEL
LIN {X 0,Y 375.318,Z 922.455,A -85,B 0,C 180,E1 -12332.146,E2 -12332.146} C_VEL
LIN {X 0,Y 375.304,Z 921.42,A -85,B 0,C 180,E1 -12333.22,E2 -12333.22} C_VEL
LIN {X 0,Y 375.339,Z 919.913,A -85,B 0,C 180,E1 -12334.295,E2 -12334.295} C_VEL
LIN {X 0,Y 375.137,Z 916.781,A -85,B 0,C 180,E1 -12335.914,E2 -12335.914} C_VEL
LIN {X 0,Y 375.146,Z 912.561,A -85,B 0,C 180,E1 -12337.535,E2 -12337.535} C_VEL
LIN {X 0,Y 375.273,Z 906.098,A -85,B 0,C 180,E1 -12339.431,E2 -12339.431} C_VEL
LIN {X 0,Y 375.637,Z 899.053,A -85,B 0,C 180,E1 -12341.056,E2 -12341.056} C_VEL
LIN {X 0,Y 376.231,Z 890.236,A -85,B 0,C 180,E1 -12342.679,E2 -12342.679} C_VEL
LIN {X 0,Y 376.822,Z 883.209,A -85,B 0,C 180,E1 -12343.756,E2 -12343.756} C_VEL
LIN {X 0,Y 377.727,Z 872.603,A -85,B 0,C 180,E1 -12345.099,E2 -12345.099} C_VEL
LIN {X 0,Y 378.652,Z 862.17,A -85,B 0,C 180,E1 -12346.165,E2 -12346.165} C_VEL
LIN {X 0,Y 379.077,Z 854.223,A -85,B 0,C 180,E1 -12346.839,E2 -12346.839} C_VEL
LIN {X 0,Y 378.284,Z 841.339,A -85,B 0,C 180,E1 -12347.762,E2 -12347.762} C_VEL
LIN {X 0,Y 377.276,Z 828.391,A -85,B 0,C 180,E1 -12348.462,E2 -12348.462} C_VEL
LIN {X 0,Y 375.839,Z 815.114,A -85,B 0,C 180,E1 -12348.977,E2 -12348.977} C_VEL
LIN {X 0,Y 375.701,Z 813.461,A -85,B 0,C 180,E1 -12349.038,E2 -12349.038} C_VEL
LIN {X 0,Y 376.314,Z 801.634,A -85,B 0,C 180,E1 -12352.511,E2 -12352.511} C_VEL
LIN {X 0,Y 377.078,Z 789.944,A -85,B 0,C 180,E1 -12355.976,E2 -12355.976} C_VEL
LIN {X 0,Y 378.039,Z 778.152,A -85,B 0,C 180,E1 -12359.535,E2 -12359.535} C_VEL
LIN {X 0,Y 379.225,Z 765.31,A -85,B 0,C 180,E1 -12363.492,E2 -12363.492} C_VEL
LIN {X 0,Y 380.358,Z 754.764,A -85,B 0,C 180,E1 -12366.828,E2 -12366.828} C_VEL
LIN {X 0,Y 380.301,Z 751.492,A -85,B 0,C 180,E1 -12367.908,E2 -12367.908} C_VEL
LIN {X 0,Y 378.479,Z 742.084,A -85,B 0,C 180,E1 -12371.232,E2 -12371.232} C_VEL
LIN {X 0,Y 376.835,Z 734.089,A -85,B 0,C 180,E1 -12374.205,E2 -12374.205} C_VEL
LIN {X 0,Y 375.947,Z 729.655,A -85,B 0,C 180,E1 -12375.967,E2 -12375.967} C_VEL
LIN {X 0,Y 375.99,Z 729.648,A -85,B 0,C 180,E1 -12380.029,E2 -12380.029} C_VEL
LIN {X 0,Y 375.965,Z 729.655,A -85,B 0,C 180,E1 -12383.496,E2 -12383.496} C_VEL
LIN {X 0,Y 375.964,Z 729.654,A -85,B 0,C 180,E1 -12385.889,E2 -12385.889} C_VEL
LIN {X 0,Y 375.966,Z 729.655,A -85,B 0,C 180,E1 -12389.687,E2 -12389.687} C_VEL
LIN {X 0,Y 375.998,Z 729.649,A -85,B 0,C 180,E1 -12392.141,E2 -12392.141} C_VEL
LIN {X 0,Y 376.007,Z 729.646,A -85,B 0,C 180,E1 -12394.539,E2 -12394.539} C_VEL
LIN {X 0,Y 375.96,Z 729.656,A -85,B 0,C 180,E1 -12398.046,E2 -12398.046} C_VEL
LIN {X 0,Y 376.025,Z 729.643,A -85,B 0,C 180,E1 -12401.474,E2 -12401.474} C_VEL
LIN {X 0,Y 376.061,Z 729.64,A -85,B 0,C 180,E1 -12404.833,E2 -12404.833} C_VEL
LIN {X 0,Y 376.052,Z 729.644,A -85,B 0,C 180,E1 -12408.137,E2 -12408.137} C_VEL
LIN {X 0,Y 376.221,Z 729.62,A -85,B 0,C 180,E1 -12411.919,E2 -12411.919} C_VEL
LIN {X 0,Y 376.169,Z 729.629,A -85,B 0,C 180,E1 -12414.64,E2 -12414.64} C_VEL
LIN {X 0,Y 376.346,Z 729.604,A -85,B 0,C 180,E1 -12417.86,E2 -12417.86} C_VEL
LIN {X 0,Y 376.485,Z 729.587,A -85,B 0,C 180,E1 -12420,E2 -12420} C_VEL
LIN {X 0,Y 376.351,Z 729.604,A -85,B 0,C 180,E1 -12422.141,E2 -12422.141} C_VEL
LIN {X 0,Y 376.21,Z 729.622,A -85,B 0,C 180,E1 -12426.485,E2 -12426.485} C_VEL
LIN {X 0,Y 376.115,Z 729.633,A -85,B 0,C 180,E1 -12429.682,E2 -12429.682} C_VEL
LIN {X 0,Y 376.092,Z 729.636,A -85,B 0,C 180,E1 -12433.658,E2 -12433.658} C_VEL
LIN {X 0,Y 376.035,Z 729.645,A -85,B 0,C 180,E1 -12437.4,E2 -12437.4} C_VEL
LIN {X 0,Y 375.98,Z 729.652,A -85,B 0,C 180,E1 -12440.832,E2 -12440.832} C_VEL
LIN {X 0,Y 375.937,Z 729.654,A -85,B 0,C 180,E1 -12444.286,E2 -12444.286} C_VEL
LIN {X 0,Y 375.928,Z 729.656,A -85,B 0,C 180,E1 -12446.659,E2 -12446.659} C_VEL
LIN {X 0,Y 375.921,Z 729.659,A -85,B 0,C 180,E1 -12449.084,E2 -12449.084} C_VEL
LIN {X 0,Y 375.959,Z 729.655,A -85,B 0,C 180,E1 -12451.562,E2 -12451.562} C_VEL
LIN {X 0,Y 375.951,Z 729.657,A -85,B 0,C 180,E1 -12455.417,E2 -12455.417} C_VEL
LIN {X 0,Y 375.936,Z 729.656,A -85,B 0,C 180,E1 -12458.263,E2 -12458.263} C_VEL
LIN {X 0,Y 375.916,Z 729.661,A -85,B 0,C 180,E1 -12461.597,E2 -12461.597} C_VEL
LIN {X 0,Y 375.921,Z 729.657,A -85,B 0,C 180,E1 -12464.73,E2 -12464.73} C_VEL
LIN {X 0,Y 375.918,Z 729.66,A -85,B 0,C 180,E1 -12467.698,E2 -12467.698} C_VEL
LIN {X 0,Y 375.935,Z 729.657,A -85,B 0,C 180,E1 -12470.534,E2 -12470.534} C_VEL
LIN {X 0,Y 375.959,Z 729.653,A -85,B 0,C 180,E1 -12473.497,E2 -12473.497} C_VEL
LIN {X 0,Y 375.959,Z 729.655,A -85,B 0,C 180,E1 -12475.888,E2 -12475.888} C_VEL
LIN {X 0,Y 375.961,Z 729.652,A -85,B 0,C 180,E1 -12479.687,E2 -12479.687} C_VEL
LIN {X 0,Y 375.918,Z 729.66,A -85,B 0,C 180,E1 -12482.135,E2 -12482.135} C_VEL
LIN {X 0,Y 375.937,Z 729.658,A -85,B 0,C 180,E1 -12484.534,E2 -12484.534} C_VEL
LIN {X 0,Y 375.976,Z 729.653,A -85,B 0,C 180,E1 -12486.887,E2 -12486.887} C_VEL
LIN {X 0,Y 375.999,Z 729.649,A -85,B 0,C 180,E1 -12490.339,E2 -12490.339} C_VEL
LIN {X 0,Y 376.026,Z 729.643,A -85,B 0,C 180,E1 -12493.719,E2 -12493.719} C_VEL
LIN {X 0,Y 376.105,Z 729.638,A -85,B 0,C 180,E1 -12497.042,E2 -12497.042} C_VEL
LIN {X 0,Y 376.109,Z 729.634,A -85,B 0,C 180,E1 -12500.318,E2 -12500.318} C_VEL
LIN {X 0,Y 376.196,Z 729.623,A -85,B 0,C 180,E1 -12503.564,E2 -12503.564} C_VEL
LIN {X 0,Y 376.34,Z 729.604,A -85,B 0,C 180,E1 -12507.86,E2 -12507.86} C_VEL
LIN {X 0,Y 376.341,Z 729.604,A -85,B 0,C 180,E1 -12512.141,E2 -12512.141} C_VEL
LIN {X 0,Y 376.201,Z 729.621,A -85,B 0,C 180,E1 -12516.436,E2 -12516.436} C_VEL
LIN {X 0,Y 376.116,Z 729.636,A -85,B 0,C 180,E1 -12519.682,E2 -12519.682} C_VEL
LIN {X 0,Y 376.093,Z 729.64,A -85,B 0,C 180,E1 -12523.658,E2 -12523.658} C_VEL
LIN {X 0,Y 376.047,Z 729.644,A -85,B 0,C 180,E1 -12527.607,E2 -12527.607} C_VEL
LIN {X 0,Y 375.982,Z 729.648,A -85,B 0,C 180,E1 -12530.832,E2 -12530.832} C_VEL
LIN {X 0,Y 375.975,Z 729.651,A -85,B 0,C 180,E1 -12534.283,E2 -12534.283} C_VEL
LIN {X 0,Y 375.938,Z 729.658,A -85,B 0,C 180,E1 -12537.864,E2 -12537.864} C_VEL
LIN {X 0,Y 375.961,Z 729.652,A -85,B 0,C 180,E1 -12541.562,E2 -12541.562} C_VEL
LIN {X 0,Y 375.961,Z 729.651,A -85,B 0,C 180,E1 -12545.416,E2 -12545.416} C_VEL
LIN {X 0,Y 375.976,Z 729.655,A -85,B 0,C 180,E1 -12548.27,E2 -12548.27} C_VEL
LIN {X 0,Y 375.986,Z 729.65,A -85,B 0,C 180,E1 -12550.015,E2 -12550.015} C_VEL
LIN {X 0,Y 375.263,Z 729.741,A -85,B 0,C 180,E1 -12550.611,E2 -12550.611} C_VEL
LIN {X 0,Y 372.377,Z 730.097,A -85,B 0,C 180,E1 -12551.541,E2 -12551.541} C_VEL
LIN {X 0,Y 369.526,Z 730.457,A -85,B 0,C 180,E1 -12552.486,E2 -12552.486} C_VEL
LIN {X 0,Y 368.876,Z 730.532,A -85,B 0,C 180,E1 -12553.097,E2 -12553.097} C_VEL
LIN {X 0,Y 368.959,Z 730.634,A -85,B 0,C 180,E1 -12554.057,E2 -12554.057} C_VEL
LIN {X 0,Y 372.304,Z 742.131,A -85,B 0,C 180,E1 -12554.988,E2 -12554.988} C_VEL
LIN {X 0,Y 374.017,Z 749.267,A -85,B 0,C 180,E1 -12555.661,E2 -12555.661} C_VEL
LIN {X 0,Y 373.283,Z 760.798,A -85,B 0,C 180,E1 -12556.776,E2 -12556.776} C_VEL
LIN {X 0,Y 372.603,Z 770.707,A -85,B 0,C 180,E1 -12557.964,E2 -12557.964} C_VEL
LIN {X 0,Y 371.857,Z 780.253,A -85,B 0,C 180,E1 -12559.372,E2 -12559.372} C_VEL
LIN {X 0,Y 371.105,Z 788.927,A -85,B 0,C 180,E1 -12560.938,E2 -12560.938} C_VEL
LIN {X 0,Y 370.468,Z 796.447,A -85,B 0,C 180,E1 -12562.622,E2 -12562.622} C_VEL
LIN {X 0,Y 369.922,Z 802.771,A -85,B 0,C 180,E1 -12564.423,E2 -12564.423} C_VEL
LIN {X 0,Y 369.511,Z 808.377,A -85,B 0,C 180,E1 -12566.525,E2 -12566.525} C_VEL
LIN {X 0,Y 369.333,Z 810.893,A -85,B 0,C 180,E1 -12567.804,E2 -12567.804} C_VEL
LIN {X 0,Y 369.175,Z 812.841,A -85,B 0,C 180,E1 -12569.069,E2 -12569.069} C_VEL
LIN {X 0,Y 369.069,Z 814.787,A -85,B 0,C 180,E1 -12571.159,E2 -12571.159} C_VEL
LIN {X 0,Y 369.213,Z 815.248,A -85,B 0,C 180,E1 -12573.464,E2 -12573.464} C_VEL
LIN {X 0,Y 369.61,Z 813.81,A -85,B 0,C 180,E1 -12575.882,E2 -12575.882} C_VEL
LIN {X 0,Y 370.049,Z 811.413,A -85,B 0,C 180,E1 -12577.676,E2 -12577.676} C_VEL
LIN {X 0,Y 370.574,Z 807.861,A -85,B 0,C 180,E1 -12579.46,E2 -12579.46} C_VEL
LIN {X 0,Y 371.28,Z 803.054,A -85,B 0,C 180,E1 -12581.228,E2 -12581.228} C_VEL
LIN {X 0,Y 372.17,Z 796.863,A -85,B 0,C 180,E1 -12582.98,E2 -12582.98} C_VEL
LIN {X 0,Y 373.214,Z 788.97,A -85,B 0,C 180,E1 -12584.714,E2 -12584.714} C_VEL
LIN {X 0,Y 374.181,Z 780.87,A -85,B 0,C 180,E1 -12586.144,E2 -12586.144} C_VEL
LIN {X 0,Y 375.179,Z 771.172,A -85,B 0,C 180,E1 -12587.538,E2 -12587.538} C_VEL
LIN {X 0,Y 376.06,Z 761.226,A -85,B 0,C 180,E1 -12588.683,E2 -12588.683} C_VEL
LIN {X 0,Y 376.569,Z 753,A -85,B 0,C 180,E1 -12589.484,E2 -12589.484} C_VEL
LIN {X 0,Y 373.689,Z 743.092,A -85,B 0,C 180,E1 -12590.528,E2 -12590.528} C_VEL
LIN {X 0,Y 370.202,Z 733.526,A -85,B 0,C 180,E1 -12591.43,E2 -12591.43} C_VEL
LIN {X 0,Y 369.112,Z 730.509,A -85,B 0,C 180,E1 -12591.708,E2 -12591.708} C_VEL
LIN {X 0,Y 369.132,Z 730.501,A -85,B 0,C 180,E1 -12594.537,E2 -12594.537} C_VEL
LIN {X 0,Y 369.318,Z 730.484,A -85,B 0,C 180,E1 -12597.819,E2 -12597.819} C_VEL
LIN {X 0,Y 369.457,Z 730.465,A -85,B 0,C 180,E1 -12600,E2 -12600} C_VEL
LIN {X 0,Y 369.317,Z 730.478,A -85,B 0,C 180,E1 -12602.181,E2 -12602.181} C_VEL
LIN {X 0,Y 369.198,Z 730.493,A -85,B 0,C 180,E1 -12606.558,E2 -12606.558} C_VEL
LIN {X 0,Y 369.068,Z 730.508,A -85,B 0,C 180,E1 -12609.868,E2 -12609.868} C_VEL
LIN {X 0,Y 369.04,Z 730.517,A -85,B 0,C 180,E1 -12613.772,E2 -12613.772} C_VEL
LIN {X 0,Y 369.004,Z 730.517,A -85,B 0,C 180,E1 -12617.768,E2 -12617.768} C_VEL
LIN {X 0,Y 368.912,Z 730.525,A -85,B 0,C 180,E1 -12621.221,E2 -12621.221} C_VEL
LIN {X 0,Y 368.958,Z 730.527,A -85,B 0,C 180,E1 -12624.775,E2 -12624.775} C_VEL
LIN {X 0,Y 368.966,Z 730.524,A -85,B 0,C 180,E1 -12627.203,E2 -12627.203} C_VEL
LIN {X 0,Y 368.932,Z 730.526,A -85,B 0,C 180,E1 -12630.953,E2 -12630.953} C_VEL
LIN {X 0,Y 368.932,Z 730.529,A -85,B 0,C 180,E1 -12635.001,E2 -12635.001} C_VEL
LIN {X 0,Y 368.911,Z 730.536,A -85,B 0,C 180,E1 -12638.64,E2 -12638.64} C_VEL
LIN {X 0,Y 368.884,Z 730.538,A -85,B 0,C 180,E1 -12642.009,E2 -12642.009} C_VEL
LIN {X 0,Y 368.921,Z 730.753,A -85,B 0,C 180,E1 -12643.124,E2 -12643.124} C_VEL
LIN {X 0,Y 370.23,Z 736.838,A -85,B 0,C 180,E1 -12646.166,E2 -12646.166} C_VEL
LIN {X 0,Y 371.862,Z 744.641,A -85,B 0,C 180,E1 -12649.602,E2 -12649.602} C_VEL
LIN {X 0,Y 372.972,Z 751.484,A -85,B 0,C 180,E1 -12652.318,E2 -12652.318} C_VEL
LIN {X 0,Y 372.246,Z 758.751,A -85,B 0,C 180,E1 -12654.851,E2 -12654.851} C_VEL
LIN {X 0,Y 371.237,Z 768.224,A -85,B 0,C 180,E1 -12657.989,E2 -12657.989} C_VEL
LIN {X 0,Y 370.251,Z 779.853,A -85,B 0,C 180,E1 -12661.67,E2 -12661.67} C_VEL
LIN {X 0,Y 369.47,Z 791.651,A -85,B 0,C 180,E1 -12665.261,E2 -12665.261} C_VEL
LIN {X 0,Y 368.818,Z 804.355,A -85,B 0,C 180,E1 -12669.022,E2 -12669.022} C_VEL
LIN {X 0,Y 368.692,Z 806.613,A -85,B 0,C 180,E1 -12669.679,E2 -12669.679} C_VEL
LIN {X 0,Y 371.059,Z 822.651,A -85,B 0,C 180,E1 -12670.443,E2 -12670.443} C_VEL
LIN {X 0,Y 371.937,Z 836.531,A -85,B 0,C 180,E1 -12671.263,E2 -12671.263} C_VEL
LIN {X 0,Y 372.164,Z 850.103,A -85,B 0,C 180,E1 -12672.276,E2 -12672.276} C_VEL
LIN {X 0,Y 372.341,Z 857.882,A -85,B 0,C 180,E1 -12672.988,E2 -12672.988} C_VEL
LIN {X 0,Y 371.083,Z 869.551,A -85,B 0,C 180,E1 -12674.202,E2 -12674.202} C_VEL
LIN {X 0,Y 370.134,Z 879.503,A -85,B 0,C 180,E1 -12675.482,E2 -12675.482} C_VEL
LIN {X 0,Y 369.442,Z 888,A -85,B 0,C 180,E1 -12676.804,E2 -12676.804} C_VEL
LIN {X 0,Y 368.703,Z 896.736,A -85,B 0,C 180,E1 -12678.454,E2 -12678.454} C_VEL
LIN {X 0,Y 368.29,Z 903.9,A -85,B 0,C 180,E1 -12680.111,E2 -12680.111} C_VEL
LIN {X 0,Y 368.088,Z 909.696,A -85,B 0,C 180,E1 -12681.767,E2 -12681.767} C_VEL
LIN {X 0,Y 368.058,Z 914.284,A -85,B 0,C 180,E1 -12683.421,E2 -12683.421} C_VEL
LIN {X 0,Y 368.101,Z 916.749,A -85,B 0,C 180,E1 -12684.522,E2 -12684.522} C_VEL
LIN {X 0,Y 368.231,Z 918.714,A -85,B 0,C 180,E1 -12685.621,E2 -12685.621} C_VEL
LIN {X 0,Y 368.256,Z 920.234,A -85,B 0,C 180,E1 -12686.718,E2 -12686.718} C_VEL
LIN {X 0,Y 368.281,Z 921.34,A -85,B 0,C 180,E1 -12687.813,E2 -12687.813} C_VEL
LIN {X 0,Y 368.325,Z 922.011,A -85,B 0,C 180,E1 -12688.907,E2 -12688.907} C_VEL
LIN {X 0,Y 368.363,Z 922.228,A -85,B 0,C 180,E1 -12690,E2 -12690} C_VEL
LIN {X 0,Y 368.326,Z 922.022,A -85,B 0,C 180,E1 -12691.093,E2 -12691.093} C_VEL
LIN {X 0,Y 368.285,Z 921.406,A -85,B 0,C 180,E1 -12692.187,E2 -12692.187} C_VEL
LIN {X 0,Y 368.268,Z 920.35,A -85,B 0,C 180,E1 -12693.282,E2 -12693.282} C_VEL
LIN {X 0,Y 368.269,Z 918.828,A -85,B 0,C 180,E1 -12694.378,E2 -12694.378} C_VEL
LIN {X 0,Y 368.089,Z 915.672,A -85,B 0,C 180,E1 -12696.028,E2 -12696.028} C_VEL
LIN {X 0,Y 368.082,Z 911.417,A -85,B 0,C 180,E1 -12697.681,E2 -12697.681} C_VEL
LIN {X 0,Y 368.241,Z 904.919,A -85,B 0,C 180,E1 -12699.613,E2 -12699.613} C_VEL
LIN {X 0,Y 368.628,Z 897.809,A -85,B 0,C 180,E1 -12701.269,E2 -12701.269} C_VEL
LIN {X 0,Y 369.271,Z 888.933,A -85,B 0,C 180,E1 -12702.922,E2 -12702.922} C_VEL
LIN {X 0,Y 370.043,Z 879.882,A -85,B 0,C 180,E1 -12704.294,E2 -12704.294} C_VEL
LIN {X 0,Y 370.879,Z 869.967,A -85,B 0,C 180,E1 -12705.525,E2 -12705.525} C_VEL
LIN {X 0,Y 371.936,Z 859.094,A -85,B 0,C 180,E1 -12706.606,E2 -12706.606} C_VEL
LIN {X 0,Y 371.904,Z 852.454,A -85,B 0,C 180,E1 -12707.174,E2 -12707.174} C_VEL
LIN {X 0,Y 371.227,Z 840.352,A -85,B 0,C 180,E1 -12708.051,E2 -12708.051} C_VEL
LIN {X 0,Y 370.198,Z 826.853,A -85,B 0,C 180,E1 -12708.792,E2 -12708.792} C_VEL
LIN {X 0,Y 368.671,Z 812.477,A -85,B 0,C 180,E1 -12709.379,E2 -12709.379} C_VEL
LIN {X 0,Y 369.206,Z 802.487,A -85,B 0,C 180,E1 -12712.378,E2 -12712.378} C_VEL
LIN {X 0,Y 370.121,Z 789.327,A -85,B 0,C 180,E1 -12716.376,E2 -12716.376} C_VEL
LIN {X 0,Y 371.101,Z 777.18,A -85,B 0,C 180,E1 -12720.123,E2 -12720.123} C_VEL
LIN {X 0,Y 372.288,Z 765.423,A -85,B 0,C 180,E1 -12723.837,E2 -12723.837} C_VEL
LIN {X 0,Y 373.41,Z 755.518,A -85,B 0,C 180,E1 -12727.033,E2 -12727.033} C_VEL
LIN {X 0,Y 373.125,Z 751.424,A -85,B 0,C 180,E1 -12728.431,E2 -12728.431} C_VEL
LIN {X 0,Y 371.201,Z 741.816,A -85,B 0,C 180,E1 -12731.918,E2 -12731.918} C_VEL
LIN {X 0,Y 369.419,Z 733.131,A -85,B 0,C 180,E1 -12735.259,E2 -12735.259} C_VEL
LIN {X 0,Y 368.888,Z 730.534,A -85,B 0,C 180,E1 -12736.312,E2 -12736.312} C_VEL
LIN {X 0,Y 368.913,Z 730.533,A -85,B 0,C 180,E1 -12739.643,E2 -12739.643} C_VEL
LIN {X 0,Y 368.903,Z 730.531,A -85,B 0,C 180,E1 -12743.144,E2 -12743.144} C_VEL
LIN {X 0,Y 368.9,Z 730.53,A -85,B 0,C 180,E1 -12746.462,E2 -12746.462} C_VEL
LIN {X 0,Y 368.93,Z 730.526,A -85,B 0,C 180,E1 -12749.047,E2 -12749.047} C_VEL
LIN {X 0,Y 368.981,Z 730.523,A -85,B 0,C 180,E1 -12751.564,E2 -12751.564} C_VEL
LIN {X 0,Y 369.001,Z 730.522,A -85,B 0,C 180,E1 -12754.02,E2 -12754.02} C_VEL
LIN {X 0,Y 368.926,Z 730.529,A -85,B 0,C 180,E1 -12757.605,E2 -12757.605} C_VEL
LIN {X 0,Y 368.984,Z 730.52,A -85,B 0,C 180,E1 -12761.107,E2 -12761.107} C_VEL
LIN {X 0,Y 369,Z 730.521,A -85,B 0,C 180,E1 -12764.535,E2 -12764.535} C_VEL
LIN {X 0,Y 369.007,Z 730.519,A -85,B 0,C 180,E1 -12767.907,E2 -12767.907} C_VEL
LIN {X 0,Y 369.168,Z 730.498,A -85,B 0,C 180,E1 -12771.869,E2 -12771.869} C_VEL
LIN {X 0,Y 369.142,Z 730.505,A -85,B 0,C 180,E1 -12774.538,E2 -12774.538} C_VEL
LIN {X 0,Y 369.31,Z 730.48,A -85,B 0,C 180,E1 -12777.819,E2 -12777.819} C_VEL
LIN {X 0,Y 369.455,Z 730.462,A -85,B 0,C 180,E1 -12780,E2 -12780} C_VEL
LIN {X 0,Y 369.316,Z 730.48,A -85,B 0,C 180,E1 -12782.181,E2 -12782.181} C_VEL
LIN {X 0,Y 369.175,Z 730.5,A -85,B 0,C 180,E1 -12786.559,E2 -12786.559} C_VEL
LIN {X 0,Y 369.065,Z 730.51,A -85,B 0,C 180,E1 -12789.868,E2 -12789.868} C_VEL
LIN {X 0,Y 369.039,Z 730.514,A -85,B 0,C 180,E1 -12793.772,E2 -12793.772} C_VEL
LIN {X 0,Y 368.993,Z 730.521,A -85,B 0,C 180,E1 -12797.743,E2 -12797.743} C_VEL
LIN {X 0,Y 368.911,Z 730.533,A -85,B 0,C 180,E1 -12801.221,E2 -12801.221} C_VEL
LIN {X 0,Y 368.912,Z 730.531,A -85,B 0,C 180,E1 -12803.875,E2 -12803.875} C_VEL
LIN {X 0,Y 368.873,Z 730.539,A -85,B 0,C 180,E1 -12807.211,E2 -12807.211} C_VEL
LIN {X 0,Y 368.931,Z 730.528,A -85,B 0,C 180,E1 -12810.954,E2 -12810.954} C_VEL
LIN {X 0,Y 368.925,Z 730.529,A -85,B 0,C 180,E1 -12815,E2 -12815} C_VEL
LIN {X 0,Y 368.878,Z 730.534,A -85,B 0,C 180,E1 -12818.634,E2 -12818.634} C_VEL
LIN {X 0,Y 368.866,Z 730.539,A -85,B 0,C 180,E1 -12822.006,E2 -12822.006} C_VEL
LIN {X 0,Y 368.874,Z 730.535,A -85,B 0,C 180,E1 -12825.175,E2 -12825.175} C_VEL
LIN {X 0,Y 368.866,Z 730.539,A -85,B 0,C 180,E1 -12828.175,E2 -12828.175} C_VEL
LIN {X 0,Y 368.877,Z 730.534,A -85,B 0,C 180,E1 -12831.366,E2 -12831.366} C_VEL
LIN {X 0,Y 368.932,Z 730.527,A -85,B 0,C 180,E1 -12835.146,E2 -12835.146} C_VEL
LIN {X 0,Y 368.897,Z 730.532,A -85,B 0,C 180,E1 -12839.043,E2 -12839.043} C_VEL
LIN {X 0,Y 368.908,Z 730.53,A -85,B 0,C 180,E1 -12841.558,E2 -12841.558} C_VEL
LIN {X 0,Y 368.888,Z 730.533,A -85,B 0,C 180,E1 -12845.22,E2 -12845.22} C_VEL
LIN {X 0,Y 368.901,Z 730.531,A -85,B 0,C 180,E1 -12847.603,E2 -12847.603} C_VEL
LIN {X 0,Y 368.957,Z 730.526,A -85,B 0,C 180,E1 -12851.106,E2 -12851.106} C_VEL
LIN {X 0,Y 368.998,Z 730.522,A -85,B 0,C 180,E1 -12854.535,E2 -12854.535} C_VEL
LIN {X 0,Y 369.06,Z 730.515,A -85,B 0,C 180,E1 -12856.79,E2 -12856.79} C_VEL
LIN {X 0,Y 369.06,Z 730.511,A -85,B 0,C 180,E1 -12860.132,E2 -12860.132} C_VEL
LIN {X 0,Y 369.157,Z 730.501,A -85,B 0,C 180,E1 -12863.441,E2 -12863.441} C_VEL
LIN {X 0,Y 369.303,Z 730.481,A -85,B 0,C 180,E1 -12867.819,E2 -12867.819} C_VEL
LIN {X 0,Y 369.305,Z 730.48,A -85,B 0,C 180,E1 -12872.181,E2 -12872.181} C_VEL
LIN {X 0,Y 369.162,Z 730.498,A -85,B 0,C 180,E1 -12876.559,E2 -12876.559} C_VEL
LIN {X 0,Y 369.066,Z 730.512,A -85,B 0,C 180,E1 -12879.868,E2 -12879.868} C_VEL
LIN {X 0,Y 369.041,Z 730.517,A -85,B 0,C 180,E1 -12883.772,E2 -12883.772} C_VEL
LIN {X 0,Y 369.005,Z 730.523,A -85,B 0,C 180,E1 -12887.768,E2 -12887.768} C_VEL
LIN {X 0,Y 368.913,Z 730.53,A -85,B 0,C 180,E1 -12891.221,E2 -12891.221} C_VEL
LIN {X 0,Y 368.929,Z 730.526,A -85,B 0,C 180,E1 -12894.778,E2 -12894.778} C_VEL
LIN {X 0,Y 368.919,Z 730.529,A -85,B 0,C 180,E1 -12898.441,E2 -12898.441} C_VEL
LIN {X 0,Y 368.913,Z 730.528,A -85,B 0,C 180,E1 -12900.987,E2 -12900.987} C_VEL
LIN {X 0,Y 368.94,Z 730.525,A -85,B 0,C 180,E1 -12904.854,E2 -12904.854} C_VEL
LIN {X 0,Y 368.91,Z 730.531,A -85,B 0,C 180,E1 -12908.64,E2 -12908.64} C_VEL
LIN {X 0,Y 368.885,Z 730.534,A -85,B 0,C 180,E1 -12912.009,E2 -12912.009} C_VEL
LIN {X 0,Y 368.876,Z 730.532,A -85,B 0,C 180,E1 -12913.097,E2 -12913.097} C_VEL
LIN {X 0,Y 368.861,Z 731.317,A -85,B 0,C 180,E1 -12913.546,E2 -12913.546} C_VEL
LIN {X 0,Y 368.749,Z 733.926,A -85,B 0,C 180,E1 -12914.039,E2 -12914.039} C_VEL
LIN {X 0,Y 368.486,Z 738.574,A -85,B 0,C 180,E1 -12914.512,E2 -12914.512} C_VEL
LIN {X 0,Y 367.482,Z 749.619,A -85,B 0,C 180,E1 -12915.377,E2 -12915.377} C_VEL
LIN {X 0,Y 366.781,Z 756.261,A -85,B 0,C 180,E1 -12915.978,E2 -12915.978} C_VEL
LIN {X 0,Y 366.063,Z 766.502,A -85,B 0,C 180,E1 -12917.099,E2 -12917.099} C_VEL
LIN {X 0,Y 365.291,Z 776.914,A -85,B 0,C 180,E1 -12918.512,E2 -12918.512} C_VEL
LIN {X 0,Y 364.475,Z 786.507,A -85,B 0,C 180,E1 -12920.122,E2 -12920.122} C_VEL
LIN {X 0,Y 363.755,Z 794.592,A -85,B 0,C 180,E1 -12921.81,E2 -12921.81} C_VEL
LIN {X 0,Y 363.175,Z 801.01,A -85,B 0,C 180,E1 -12923.483,E2 -12923.483} C_VEL
LIN {X 0,Y 362.707,Z 806.094,A -85,B 0,C 180,E1 -12925.137,E2 -12925.137} C_VEL
LIN {X 0,Y 362.404,Z 810.71,A -85,B 0,C 180,E1 -12927.112,E2 -12927.112} C_VEL
LIN {X 0,Y 362.181,Z 813.271,A -85,B 0,C 180,E1 -12928.629,E2 -12928.629} C_VEL
LIN {X 0,Y 362.121,Z 814.616,A -85,B 0,C 180,E1 -12929.695,E2 -12929.695} C_VEL
LIN {X 0,Y 362.058,Z 815.709,A -85,B 0,C 180,E1 -12930.969,E2 -12930.969} C_VEL
LIN {X 0,Y 362.072,Z 816.284,A -85,B 0,C 180,E1 -12932.234,E2 -12932.234} C_VEL
LIN {X 0,Y 362.215,Z 816.337,A -85,B 0,C 180,E1 -12933.495,E2 -12933.495} C_VEL
LIN {X 0,Y 362.556,Z 815.216,A -85,B 0,C 180,E1 -12935.655,E2 -12935.655} C_VEL
LIN {X 0,Y 362.921,Z 813.461,A -85,B 0,C 180,E1 -12937.213,E2 -12937.213} C_VEL
LIN {X 0,Y 363.469,Z 810.33,A -85,B 0,C 180,E1 -12939.04,E2 -12939.04} C_VEL
LIN {X 0,Y 364.213,Z 805.577,A -85,B 0,C 180,E1 -12941.002,E2 -12941.002} C_VEL
LIN {X 0,Y 365.178,Z 799.193,A -85,B 0,C 180,E1 -12942.933,E2 -12942.933} C_VEL
LIN {X 0,Y 366.284,Z 791.659,A -85,B 0,C 180,E1 -12944.703,E2 -12944.703} C_VEL
LIN {X 0,Y 367.238,Z 783.928,A -85,B 0,C 180,E1 -12946.159,E2 -12946.159} C_VEL
LIN {X 0,Y 368.286,Z 775.144,A -85,B 0,C 180,E1 -12947.508,E2 -12947.508} C_VEL
LIN {X 0,Y 369.243,Z 765.268,A -85,B 0,C 180,E1 -12948.75,E2 -12948.75} C_VEL
LIN {X 0,Y 369.944,Z 754.259,A -85,B 0,C 180,E1 -12949.879,E2 -12949.879} C_VEL
LIN {X 0,Y 366.91,Z 744.336,A -85,B 0,C 180,E1 -12950.965,E2 -12950.965} C_VEL
LIN {X 0,Y 363.228,Z 734.481,A -85,B 0,C 180,E1 -12951.937,E2 -12951.937} C_VEL
LIN {X 0,Y 362.08,Z 731.381,A -85,B 0,C 180,E1 -12952.226,E2 -12952.226} C_VEL
LIN {X 0,Y 362.103,Z 731.376,A -85,B 0,C 180,E1 -12954.431,E2 -12954.431} C_VEL
LIN {X 0,Y 362.281,Z 731.36,A -85,B 0,C 180,E1 -12957.776,E2 -12957.776} C_VEL
LIN {X 0,Y 362.405,Z 731.344,A -85,B 0,C 180,E1 -12960,E2 -12960} C_VEL
LIN {X 0,Y 362.281,Z 731.354,A -85,B 0,C 180,E1 -12962.223,E2 -12962.223} C_VEL
LIN {X 0,Y 362.161,Z 731.371,A -85,B 0,C 180,E1 -12966.686,E2 -12966.686} C_VEL
LIN {X 0,Y 362.033,Z 731.387,A -85,B 0,C 180,E1 -12970.062,E2 -12970.062} C_VEL
LIN {X 0,Y 362.001,Z 731.394,A -85,B 0,C 180,E1 -12973.899,E2 -12973.899} C_VEL
LIN {X 0,Y 361.97,Z 731.392,A -85,B 0,C 180,E1 -12977.938,E2 -12977.938} C_VEL
LIN {X 0,Y 361.864,Z 731.404,A -85,B 0,C 180,E1 -12981.655,E2 -12981.655} C_VEL
LIN {X 0,Y 361.93,Z 731.401,A -85,B 0,C 180,E1 -12985.29,E2 -12985.29} C_VEL
LIN {X 0,Y 361.911,Z 731.404,A -85,B 0,C 180,E1 -12987.779,E2 -12987.779} C_VEL
LIN {X 0,Y 361.84,Z 731.411,A -85,B 0,C 180,E1 -12991.629,E2 -12991.629} C_VEL
LIN {X 0,Y 361.877,Z 731.408,A -85,B 0,C 180,E1 -12995.345,E2 -12995.345} C_VEL
LIN {X 0,Y 361.872,Z 731.413,A -85,B 0,C 180,E1 -12999.027,E2 -12999.027} C_VEL
LIN {X 0,Y 361.898,Z 731.604,A -85,B 0,C 180,E1 -13002.442,E2 -13002.442} C_VEL
LIN {X 0,Y 363.212,Z 737.926,A -85,B 0,C 180,E1 -13005.72,E2 -13005.72} C_VEL
LIN {X 0,Y 364.716,Z 745.216,A -85,B 0,C 180,E1 -13009.067,E2 -13009.067} C_VEL
LIN {X 0,Y 365.953,Z 752.211,A -85,B 0,C 180,E1 -13011.943,E2 -13011.943} C_VEL
LIN {X 0,Y 365.787,Z 756.255,A -85,B 0,C 180,E1 -13013.443,E2 -13013.443} C_VEL
LIN {X 0,Y 364.465,Z 767.529,A -85,B 0,C 180,E1 -13017.321,E2 -13017.321} C_VEL
LIN {X 0,Y 363.342,Z 779.077,A -85,B 0,C 180,E1 -13021.081,E2 -13021.081} C_VEL
LIN {X 0,Y 362.524,Z 790.781,A -85,B 0,C 180,E1 -13024.754,E2 -13024.754} C_VEL
LIN {X 0,Y 361.762,Z 804.197,A -85,B 0,C 180,E1 -13028.829,E2 -13028.829} C_VEL
LIN {X 0,Y 361.725,Z 805.614,A -85,B 0,C 180,E1 -13029.199,E2 -13029.199} C_VEL
LIN {X 0,Y 364.005,Z 820.375,A -85,B 0,C 180,E1 -13029.906,E2 -13029.906} C_VEL
LIN {X 0,Y 365.008,Z 832.762,A -85,B 0,C 180,E1 -13030.642,E2 -13030.642} C_VEL
LIN {X 0,Y 365.241,Z 844.927,A -85,B 0,C 180,E1 -13031.524,E2 -13031.524} C_VEL
LIN {X 0,Y 365.503,Z 857.339,A -85,B 0,C 180,E1 -13032.66,E2 -13032.66} C_VEL
LIN {X 0,Y 364.228,Z 868.911,A -85,B 0,C 180,E1 -13033.896,E2 -13033.896} C_VEL
LIN {X 0,Y 363.224,Z 878.396,A -85,B 0,C 180,E1 -13035.145,E2 -13035.145} C_VEL
LIN {X 0,Y 362.485,Z 887.192,A -85,B 0,C 180,E1 -13036.546,E2 -13036.546} C_VEL
LIN {X 0,Y 361.705,Z 895.879,A -85,B 0,C 180,E1 -13038.228,E2 -13038.228} C_VEL
LIN {X 0,Y 361.229,Z 902.983,A -85,B 0,C 180,E1 -13039.915,E2 -13039.915} C_VEL
LIN {X 0,Y 361.002,Z 908.739,A -85,B 0,C 180,E1 -13041.604,E2 -13041.604} C_VEL
LIN {X 0,Y 360.989,Z 913.312,A -85,B 0,C 180,E1 -13043.292,E2 -13043.292} C_VEL
LIN {X 0,Y 361.034,Z 915.758,A -85,B 0,C 180,E1 -13044.414,E2 -13044.414} C_VEL
LIN {X 0,Y 361.169,Z 917.715,A -85,B 0,C 180,E1 -13045.536,E2 -13045.536} C_VEL
LIN {X 0,Y 361.213,Z 919.235,A -85,B 0,C 180,E1 -13046.654,E2 -13046.654} C_VEL
LIN {X 0,Y 361.24,Z 920.334,A -85,B 0,C 180,E1 -13047.77,E2 -13047.77} C_VEL
LIN {X 0,Y 361.293,Z 920.982,A -85,B 0,C 180,E1 -13048.885,E2 -13048.885} C_VEL
LIN {X 0,Y 361.339,Z 921.189,A -85,B 0,C 180,E1 -13050,E2 -13050} C_VEL
LIN {X 0,Y 361.298,Z 920.975,A -85,B 0,C 180,E1 -13051.114,E2 -13051.114} C_VEL
LIN {X 0,Y 361.252,Z 920.349,A -85,B 0,C 180,E1 -13052.23,E2 -13052.23} C_VEL
LIN {X 0,Y 361.231,Z 919.261,A -85,B 0,C 180,E1 -13053.346,E2 -13053.346} C_VEL
LIN {X 0,Y 361.122,Z 916.795,A -85,B 0,C 180,E1 -13055.024,E2 -13055.024} C_VEL
LIN {X 0,Y 361.046,Z 912.757,A -85,B 0,C 180,E1 -13056.903,E2 -13056.903} C_VEL
LIN {X 0,Y 361.084,Z 906.728,A -85,B 0,C 180,E1 -13058.958,E2 -13058.958} C_VEL
LIN {X 0,Y 361.329,Z 900.312,A -85,B 0,C 180,E1 -13060.648,E2 -13060.648} C_VEL
LIN {X 0,Y 361.919,Z 892.299,A -85,B 0,C 180,E1 -13062.334,E2 -13062.334} C_VEL
LIN {X 0,Y 362.638,Z 884.46,A -85,B 0,C 180,E1 -13063.687,E2 -13063.687} C_VEL
LIN {X 0,Y 363.248,Z 876.617,A -85,B 0,C 180,E1 -13064.825,E2 -13064.825} C_VEL
LIN {X 0,Y 364.188,Z 865.899,A -85,B 0,C 180,E1 -13066.105,E2 -13066.105} C_VEL
LIN {X 0,Y 365.073,Z 855.89,A -85,B 0,C 180,E1 -13067.072,E2 -13067.072} C_VEL
LIN {X 0,Y 364.412,Z 843.895,A -85,B 0,C 180,E1 -13068.045,E2 -13068.045} C_VEL
LIN {X 0,Y 363.532,Z 830.577,A -85,B 0,C 180,E1 -13068.871,E2 -13068.871} C_VEL
LIN {X 0,Y 362.194,Z 816.883,A -85,B 0,C 180,E1 -13069.5,E2 -13069.5} C_VEL
LIN {X 0,Y 361.622,Z 811.597,A -85,B 0,C 180,E1 -13069.698,E2 -13069.698} C_VEL
LIN {X 0,Y 362.181,Z 801.408,A -85,B 0,C 180,E1 -13072.836,E2 -13072.836} C_VEL
LIN {X 0,Y 363.055,Z 789.803,A -85,B 0,C 180,E1 -13076.438,E2 -13076.438} C_VEL
LIN {X 0,Y 364.045,Z 778.11,A -85,B 0,C 180,E1 -13080.128,E2 -13080.128} C_VEL
LIN {X 0,Y 365.38,Z 765.493,A -85,B 0,C 180,E1 -13084.198,E2 -13084.198} C_VEL
LIN {X 0,Y 366.452,Z 756.496,A -85,B 0,C 180,E1 -13087.166,E2 -13087.166} C_VEL
LIN {X 0,Y 366.054,Z 752.212,A -85,B 0,C 180,E1 -13088.674,E2 -13088.674} C_VEL
LIN {X 0,Y 364.265,Z 743.297,A -85,B 0,C 180,E1 -13091.965,E2 -13091.965} C_VEL
LIN {X 0,Y 362.262,Z 733.341,A -85,B 0,C 180,E1 -13095.874,E2 -13095.874} C_VEL
LIN {X 0,Y 361.853,Z 731.411,A -85,B 0,C 180,E1 -13096.751,E2 -13096.751} C_VEL
LIN {X 0,Y 361.856,Z 731.409,A -85,B 0,C 180,E1 -13100.139,E2 -13100.139} C_VEL
LIN {X 0,Y 361.869,Z 731.406,A -85,B 0,C 180,E1 -13102.982,E2 -13102.982} C_VEL
LIN {X 0,Y 361.862,Z 731.406,A -85,B 0,C 180,E1 -13106.63,E2 -13106.63} C_VEL
LIN {X 0,Y 361.876,Z 731.41,A -85,B 0,C 180,E1 -13109.672,E2 -13109.672} C_VEL
LIN {X 0,Y 361.956,Z 731.397,A -85,B 0,C 180,E1 -13113.475,E2 -13113.475} C_VEL
LIN {X 0,Y 361.884,Z 731.404,A -85,B 0,C 180,E1 -13117.144,E2 -13117.144} C_VEL
LIN {X 0,Y 361.923,Z 731.4,A -85,B 0,C 180,E1 -13120.724,E2 -13120.724} C_VEL
LIN {X 0,Y 361.948,Z 731.401,A -85,B 0,C 180,E1 -13124.226,E2 -13124.226} C_VEL
LIN {X 0,Y 362.001,Z 731.393,A -85,B 0,C 180,E1 -13126.528,E2 -13126.528} C_VEL
LIN {X 0,Y 362.033,Z 731.388,A -85,B 0,C 180,E1 -13129.938,E2 -13129.938} C_VEL
LIN {X 0,Y 362.164,Z 731.37,A -85,B 0,C 180,E1 -13133.314,E2 -13133.314} C_VEL
LIN {X 0,Y 362.273,Z 731.356,A -85,B 0,C 180,E1 -13137.777,E2 -13137.777} C_VEL
LIN {X 0,Y 362.404,Z 731.34,A -85,B 0,C 180,E1 -13140,E2 -13140} C_VEL
LIN {X 0,Y 362.28,Z 731.357,A -85,B 0,C 180,E1 -13142.224,E2 -13142.224} C_VEL
LIN {X 0,Y 362.137,Z 731.378,A -85,B 0,C 180,E1 -13146.687,E2 -13146.687} C_VEL
LIN {X 0,Y 362.002,Z 731.39,A -85,B 0,C 180,E1 -13150.063,E2 -13150.063} C_VEL
LIN {X 0,Y 362,Z 731.39,A -85,B 0,C 180,E1 -13153.899,E2 -13153.899} C_VEL
LIN {X 0,Y 361.93,Z 731.403,A -85,B 0,C 180,E1 -13156.934,E2 -13156.934} C_VEL
LIN {X 0,Y 361.888,Z 731.404,A -85,B 0,C 180,E1 -13160.461,E2 -13160.461} C_VEL
LIN {X 0,Y 361.862,Z 731.408,A -85,B 0,C 180,E1 -13164.101,E2 -13164.101} C_VEL
LIN {X 0,Y 361.847,Z 731.412,A -85,B 0,C 180,E1 -13167.784,E2 -13167.784} C_VEL
LIN {X 0,Y 361.849,Z 731.413,A -85,B 0,C 180,E1 -13171.285,E2 -13171.285} C_VEL
LIN {X 0,Y 361.852,Z 731.409,A -85,B 0,C 180,E1 -13174.281,E2 -13174.281} C_VEL
LIN {X 0,Y 361.859,Z 731.41,A -85,B 0,C 180,E1 -13177.222,E2 -13177.222} C_VEL
LIN {X 0,Y 361.812,Z 731.414,A -85,B 0,C 180,E1 -13180.751,E2 -13180.751} C_VEL
LIN {X 0,Y 361.813,Z 731.416,A -85,B 0,C 180,E1 -13184.37,E2 -13184.37} C_VEL
LIN {X 0,Y 361.827,Z 731.414,A -85,B 0,C 180,E1 -13187.57,E2 -13187.57} C_VEL
LIN {X 0,Y 361.843,Z 731.411,A -85,B 0,C 180,E1 -13191.572,E2 -13191.572} C_VEL
LIN {X 0,Y 361.871,Z 731.408,A -85,B 0,C 180,E1 -13194.657,E2 -13194.657} C_VEL
LIN {X 0,Y 361.839,Z 731.414,A -85,B 0,C 180,E1 -13198.371,E2 -13198.371} C_VEL
LIN {X 0,Y 361.868,Z 731.408,A -85,B 0,C 180,E1 -13200.952,E2 -13200.952} C_VEL
LIN {X 0,Y 361.862,Z 731.411,A -85,B 0,C 180,E1 -13204.705,E2 -13204.705} C_VEL
LIN {X 0,Y 361.857,Z 731.412,A -85,B 0,C 180,E1 -13208.345,E2 -13208.345} C_VEL
LIN {X 0,Y 361.923,Z 731.401,A -85,B 0,C 180,E1 -13212.085,E2 -13212.085} C_VEL
LIN {X 0,Y 361.964,Z 731.396,A -85,B 0,C 180,E1 -13215.38,E2 -13215.38} C_VEL
LIN {X 0,Y 361.966,Z 731.398,A -85,B 0,C 180,E1 -13218.804,E2 -13218.804} C_VEL
LIN {X 0,Y 362.08,Z 731.38,A -85,B 0,C 180,E1 -13222.191,E2 -13222.191} C_VEL
LIN {X 0,Y 362.09,Z 731.38,A -85,B 0,C 180,E1 -13224.431,E2 -13224.431} C_VEL
LIN {X 0,Y 362.266,Z 731.357,A -85,B 0,C 180,E1 -13227.776,E2 -13227.776} C_VEL
LIN {X 0,Y 362.177,Z 731.372,A -85,B 0,C 180,E1 -13231.112,E2 -13231.112} C_VEL
LIN {X 0,Y 362.268,Z 731.356,A -85,B 0,C 180,E1 -13232.224,E2 -13232.224} C_VEL
LIN {X 0,Y 362.125,Z 731.375,A -85,B 0,C 180,E1 -13236.687,E2 -13236.687} C_VEL
LIN {X 0,Y 362.003,Z 731.39,A -85,B 0,C 180,E1 -13240.063,E2 -13240.063} C_VEL
LIN {X 0,Y 362.001,Z 731.392,A -85,B 0,C 180,E1 -13243.899,E2 -13243.899} C_VEL
LIN {X 0,Y 361.971,Z 731.397,A -85,B 0,C 180,E1 -13247.939,E2 -13247.939} C_VEL
LIN {X 0,Y 361.858,Z 731.412,A -85,B 0,C 180,E1 -13251.655,E2 -13251.655} C_VEL
LIN {X 0,Y 361.886,Z 731.405,A -85,B 0,C 180,E1 -13255.293,E2 -13255.293} C_VEL
LIN {X 0,Y 361.858,Z 731.407,A -85,B 0,C 180,E1 -13259.074,E2 -13259.074} C_VEL
LIN {X 0,Y 361.852,Z 731.408,A -85,B 0,C 180,E1 -13262.945,E2 -13262.945} C_VEL
LIN {X 0,Y 361.871,Z 731.407,A -85,B 0,C 180,E1 -13265.637,E2 -13265.637} C_VEL
LIN {X 0,Y 361.871,Z 731.405,A -85,B 0,C 180,E1 -13269.026,E2 -13269.026} C_VEL
LIN {X 0,Y 361.84,Z 731.411,A -85,B 0,C 180,E1 -13272.829,E2 -13272.829} C_VEL
LIN {X 0,Y 361.873,Z 731.462,A -85,B 0,C 180,E1 -13273.757,E2 -13273.757} C_VEL
LIN {X 0,Y 365.218,Z 743.02,A -85,B 0,C 180,E1 -13274.712,E2 -13274.712} C_VEL
LIN {X 0,Y 367.062,Z 749.844,A -85,B 0,C 180,E1 -13275.376,E2 -13275.376} C_VEL
LIN {X 0,Y 366.781,Z 756.261,A -85,B 0,C 180,E1 -13275.978,E2 -13275.978} C_VEL
LIN {X 0,Y 365.764,Z 761.235,A -85,B 0,C 180,E1 -13276.454,E2 -13276.454} C_VEL
LIN {X 0,Y 362.495,Z 769.141,A -85,B 0,C 180,E1 -13277.244,E2 -13277.244} C_VEL
LIN {X 0,Y 359.193,Z 776.576,A -85,B 0,C 180,E1 -13278.14,E2 -13278.14} C_VEL
LIN {X 0,Y 358.14,Z 780.809,A -85,B 0,C 180,E1 -13278.776,E2 -13278.776} C_VEL
LIN {X 0,Y 357.312,Z 789.513,A -85,B 0,C 180,E1 -13280.351,E2 -13280.351} C_VEL
LIN {X 0,Y 356.612,Z 797.037,A -85,B 0,C 180,E1 -13282.028,E2 -13282.028} C_VEL
LIN {X 0,Y 356.109,Z 803.069,A -85,B 0,C 180,E1 -13283.696,E2 -13283.696} C_VEL
LIN {X 0,Y 355.591,Z 808.599,A -85,B 0,C 180,E1 -13285.641,E2 -13285.641} C_VEL
LIN {X 0,Y 355.296,Z 812.887,A -85,B 0,C 180,E1 -13287.718,E2 -13287.718} C_VEL
LIN {X 0,Y 355.146,Z 814.879,A -85,B 0,C 180,E1 -13289.035,E2 -13289.035} C_VEL
LIN {X 0,Y 355.035,Z 816.461,A -85,B 0,C 180,E1 -13290.575,E2 -13290.575} C_VEL
LIN {X 0,Y 355.053,Z 817.135,A -85,B 0,C 180,E1 -13291.636,E2 -13291.636} C_VEL
LIN {X 0,Y 355.137,Z 817.437,A -85,B 0,C 180,E1 -13292.941,E2 -13292.941} C_VEL
LIN {X 0,Y 355.284,Z 817.27,A -85,B 0,C 180,E1 -13294.202,E2 -13294.202} C_VEL
LIN {X 0,Y 355.509,Z 816.572,A -85,B 0,C 180,E1 -13295.471,E2 -13295.471} C_VEL
LIN {X 0,Y 355.812,Z 815.382,A -85,B 0,C 180,E1 -13296.731,E2 -13296.731} C_VEL
LIN {X 0,Y 356.37,Z 812.621,A -85,B 0,C 180,E1 -13298.63,E2 -13298.63} C_VEL
LIN {X 0,Y 357.034,Z 808.771,A -85,B 0,C 180,E1 -13300.449,E2 -13300.449} C_VEL
LIN {X 0,Y 357.906,Z 803.54,A -85,B 0,C 180,E1 -13302.28,E2 -13302.28} C_VEL
LIN {X 0,Y 358.939,Z 796.888,A -85,B 0,C 180,E1 -13304.09,E2 -13304.09} C_VEL
LIN {X 0,Y 359.966,Z 790.017,A -85,B 0,C 180,E1 -13305.585,E2 -13305.585} C_VEL
LIN {X 0,Y 361.026,Z 781.642,A -85,B 0,C 180,E1 -13307.079,E2 -13307.079} C_VEL
LIN {X 0,Y 362.208,Z 771.461,A -85,B 0,C 180,E1 -13308.528,E2 -13308.528} C_VEL
LIN {X 0,Y 363.149,Z 761.421,A -85,B 0,C 180,E1 -13309.687,E2 -13309.687} C_VEL
LIN {X 0,Y 363.501,Z 757.05,A -85,B 0,C 180,E1 -13310.119,E2 -13310.119} C_VEL
LIN {X 0,Y 360.51,Z 746.732,A -85,B 0,C 180,E1 -13311.314,E2 -13311.314} C_VEL
LIN {X 0,Y 357.307,Z 737.946,A -85,B 0,C 180,E1 -13312.229,E2 -13312.229} C_VEL
LIN {X 0,Y 355.523,Z 734.083,A -85,B 0,C 180,E1 -13312.622,E2 -13312.622} C_VEL
LIN {X 0,Y 355.053,Z 732.257,A -85,B 0,C 180,E1 -13312.789,E2 -13312.789} C_VEL
LIN {X 0,Y 355.076,Z 732.252,A -85,B 0,C 180,E1 -13314.32,E2 -13314.32} C_VEL
LIN {X 0,Y 355.244,Z 732.236,A -85,B 0,C 180,E1 -13317.732,E2 -13317.732} C_VEL
LIN {X 0,Y 355.356,Z 732.222,A -85,B 0,C 180,E1 -13320,E2 -13320} C_VEL
LIN {X 0,Y 355.244,Z 732.23,A -85,B 0,C 180,E1 -13322.268,E2 -13322.268} C_VEL
LIN {X 0,Y 355.125,Z 732.247,A -85,B 0,C 180,E1 -13326.819,E2 -13326.819} C_VEL
LIN {X 0,Y 354.98,Z 732.269,A -85,B 0,C 180,E1 -13330.264,E2 -13330.264} C_VEL
LIN {X 0,Y 354.946,Z 732.271,A -85,B 0,C 180,E1 -13334.019,E2 -13334.019} C_VEL
LIN {X 0,Y 354.925,Z 732.269,A -85,B 0,C 180,E1 -13338.108,E2 -13338.108} C_VEL
LIN {X 0,Y 354.819,Z 732.286,A -85,B 0,C 180,E1 -13342.107,E2 -13342.107} C_VEL
LIN {X 0,Y 354.901,Z 732.276,A -85,B 0,C 180,E1 -13345.827,E2 -13345.827} C_VEL
LIN {X 0,Y 354.82,Z 732.286,A -85,B 0,C 180,E1 -13349.682,E2 -13349.682} C_VEL
LIN {X 0,Y 354.808,Z 732.288,A -85,B 0,C 180,E1 -13353.702,E2 -13353.702} C_VEL
LIN {X 0,Y 354.801,Z 732.294,A -85,B 0,C 180,E1 -13356.459,E2 -13356.459} C_VEL
LIN {X 0,Y 354.826,Z 732.293,A -85,B 0,C 180,E1 -13359.423,E2 -13359.423} C_VEL
LIN {X 0,Y 354.825,Z 732.458,A -85,B 0,C 180,E1 -13361.699,E2 -13361.699} C_VEL
LIN {X 0,Y 356.24,Z 738.982,A -85,B 0,C 180,E1 -13365.253,E2 -13365.253} C_VEL
LIN {X 0,Y 357.53,Z 745.43,A -85,B 0,C 180,E1 -13368.329,E2 -13368.329} C_VEL
LIN {X 0,Y 358.794,Z 752.025,A -85,B 0,C 180,E1 -13371.184,E2 -13371.184} C_VEL
LIN {X 0,Y 359.057,Z 755.713,A -85,B 0,C 180,E1 -13372.643,E2 -13372.643} C_VEL
LIN {X 0,Y 357.861,Z 765.296,A -85,B 0,C 180,E1 -13376.076,E2 -13376.076} C_VEL
LIN {X 0,Y 356.483,Z 778.3,A -85,B 0,C 180,E1 -13380.47,E2 -13380.47} C_VEL
LIN {X 0,Y 355.554,Z 789.94,A -85,B 0,C 180,E1 -13384.223,E2 -13384.223} C_VEL
LIN {X 0,Y 354.78,Z 803.078,A -85,B 0,C 180,E1 -13388.325,E2 -13388.325} C_VEL
LIN {X 0,Y 354.71,Z 804.066,A -85,B 0,C 180,E1 -13388.628,E2 -13388.628} C_VEL
LIN {X 0,Y 357.175,Z 819.904,A -85,B 0,C 180,E1 -13389.445,E2 -13389.445} C_VEL
LIN {X 0,Y 358.237,Z 832.338,A -85,B 0,C 180,E1 -13390.22,E2 -13390.22} C_VEL
LIN {X 0,Y 358.434,Z 844.99,A -85,B 0,C 180,E1 -13391.181,E2 -13391.181} C_VEL
LIN {X 0,Y 358.546,Z 856.945,A -85,B 0,C 180,E1 -13392.313,E2 -13392.313} C_VEL
LIN {X 0,Y 357.688,Z 865.967,A -85,B 0,C 180,E1 -13393.3,E2 -13393.3} C_VEL
LIN {X 0,Y 356.482,Z 875.697,A -85,B 0,C 180,E1 -13394.564,E2 -13394.564} C_VEL
LIN {X 0,Y 355.549,Z 885.309,A -85,B 0,C 180,E1 -13396.082,E2 -13396.082} C_VEL
LIN {X 0,Y 354.786,Z 893.715,A -85,B 0,C 180,E1 -13397.705,E2 -13397.705} C_VEL
LIN {X 0,Y 354.195,Z 901,A -85,B 0,C 180,E1 -13399.424,E2 -13399.424} C_VEL
LIN {X 0,Y 353.94,Z 907.825,A -85,B 0,C 180,E1 -13401.435,E2 -13401.435} C_VEL
LIN {X 0,Y 353.937,Z 913.13,A -85,B 0,C 180,E1 -13403.503,E2 -13403.503} C_VEL
LIN {X 0,Y 354.109,Z 916.724,A -85,B 0,C 180,E1 -13405.446,E2 -13405.446} C_VEL
LIN {X 0,Y 354.171,Z 918.237,A -85,B 0,C 180,E1 -13406.587,E2 -13406.587} C_VEL
LIN {X 0,Y 354.199,Z 919.326,A -85,B 0,C 180,E1 -13407.726,E2 -13407.726} C_VEL
LIN {X 0,Y 354.262,Z 919.953,A -85,B 0,C 180,E1 -13408.863,E2 -13408.863} C_VEL
LIN {X 0,Y 354.314,Z 920.155,A -85,B 0,C 180,E1 -13410,E2 -13410} C_VEL
LIN {X 0,Y 354.269,Z 919.93,A -85,B 0,C 180,E1 -13411.137,E2 -13411.137} C_VEL
LIN {X 0,Y 354.219,Z 919.287,A -85,B 0,C 180,E1 -13412.274,E2 -13412.274} C_VEL
LIN {X 0,Y 354.19,Z 918.172,A -85,B 0,C 180,E1 -13413.413,E2 -13413.413} C_VEL
LIN {X 0,Y 354.071,Z 915.675,A -85,B 0,C 180,E1 -13415.124,E2 -13415.124} C_VEL
LIN {X 0,Y 353.984,Z 911.891,A -85,B 0,C 180,E1 -13416.926,E2 -13416.926} C_VEL
LIN {X 0,Y 353.997,Z 907.371,A -85,B 0,C 180,E1 -13418.563,E2 -13418.563} C_VEL
LIN {X 0,Y 354.247,Z 900.226,A -85,B 0,C 180,E1 -13420.574,E2 -13420.574} C_VEL
LIN {X 0,Y 354.803,Z 892.487,A -85,B 0,C 180,E1 -13422.295,E2 -13422.295} C_VEL
LIN {X 0,Y 355.589,Z 883.335,A -85,B 0,C 180,E1 -13423.923,E2 -13423.923} C_VEL
LIN {X 0,Y 356.576,Z 872.844,A -85,B 0,C 180,E1 -13425.431,E2 -13425.431} C_VEL
LIN {X 0,Y 357.495,Z 863.098,A -85,B 0,C 180,E1 -13426.562,E2 -13426.562} C_VEL
LIN {X 0,Y 358.005,Z 855.8,A -85,B 0,C 180,E1 -13427.273,E2 -13427.273} C_VEL
LIN {X 0,Y 357.41,Z 843.063,A -85,B 0,C 180,E1 -13428.338,E2 -13428.338} C_VEL
LIN {X 0,Y 356.499,Z 829.965,A -85,B 0,C 180,E1 -13429.173,E2 -13429.173} C_VEL
LIN {X 0,Y 355.128,Z 815.897,A -85,B 0,C 180,E1 -13429.833,E2 -13429.833} C_VEL
LIN {X 0,Y 354.597,Z 810.705,A -85,B 0,C 180,E1 -13430.03,E2 -13430.03} C_VEL
LIN {X 0,Y 355.171,Z 800.283,A -85,B 0,C 180,E1 -13433.313,E2 -13433.313} C_VEL
LIN {X 0,Y 356.096,Z 788.719,A -85,B 0,C 180,E1 -13436.996,E2 -13436.996} C_VEL
LIN {X 0,Y 357.035,Z 778.462,A -85,B 0,C 180,E1 -13440.314,E2 -13440.314} C_VEL
LIN {X 0,Y 358.251,Z 767.397,A -85,B 0,C 180,E1 -13443.951,E2 -13443.951} C_VEL
LIN {X 0,Y 359.474,Z 757.433,A -85,B 0,C 180,E1 -13447.306,E2 -13447.306} C_VEL
LIN {X 0,Y 359.039,Z 753.312,A -85,B 0,C 180,E1 -13448.784,E2 -13448.784} C_VEL
LIN {X 0,Y 357.055,Z 743.296,A -85,B 0,C 180,E1 -13452.587,E2 -13452.587} C_VEL
LIN {X 0,Y 354.969,Z 733.129,A -85,B 0,C 180,E1 -13456.695,E2 -13456.695} C_VEL
LIN {X 0,Y 354.793,Z 732.291,A -85,B 0,C 180,E1 -13457.132,E2 -13457.132} C_VEL
LIN {X 0,Y 354.816,Z 732.287,A -85,B 0,C 180,E1 -13460.666,E2 -13460.666} C_VEL
LIN {X 0,Y 354.823,Z 732.284,A -85,B 0,C 180,E1 -13464.301,E2 -13464.301} C_VEL
LIN {X 0,Y 354.789,Z 732.293,A -85,B 0,C 180,E1 -13467.667,E2 -13467.667} C_VEL
LIN {X 0,Y 354.87,Z 732.278,A -85,B 0,C 180,E1 -13470.621,E2 -13470.621} C_VEL
LIN {X 0,Y 354.9,Z 732.278,A -85,B 0,C 180,E1 -13474.173,E2 -13474.173} C_VEL
LIN {X 0,Y 354.828,Z 732.288,A -85,B 0,C 180,E1 -13477.894,E2 -13477.894} C_VEL
LIN {X 0,Y 354.925,Z 732.274,A -85,B 0,C 180,E1 -13481.891,E2 -13481.891} C_VEL
LIN {X 0,Y 354.945,Z 732.272,A -85,B 0,C 180,E1 -13485.981,E2 -13485.981} C_VEL
LIN {X 0,Y 354.98,Z 732.265,A -85,B 0,C 180,E1 -13489.736,E2 -13489.736} C_VEL
LIN {X 0,Y 355.127,Z 732.246,A -85,B 0,C 180,E1 -13493.181,E2 -13493.181} C_VEL
LIN {X 0,Y 355.236,Z 732.232,A -85,B 0,C 180,E1 -13497.732,E2 -13497.732} C_VEL
LIN {X 0,Y 355.354,Z 732.218,A -85,B 0,C 180,E1 -13500,E2 -13500} C_VEL
LIN {X 0,Y 355.242,Z 732.233,A -85,B 0,C 180,E1 -13502.268,E2 -13502.268} C_VEL
LIN {X 0,Y 355.101,Z 732.254,A -85,B 0,C 180,E1 -13506.82,E2 -13506.82} C_VEL
LIN {X 0,Y 354.958,Z 732.268,A -85,B 0,C 180,E1 -13510.265,E2 -13510.265} C_VEL
LIN {X 0,Y 354.945,Z 732.269,A -85,B 0,C 180,E1 -13514.019,E2 -13514.019} C_VEL
LIN {X 0,Y 354.892,Z 732.275,A -85,B 0,C 180,E1 -13518.092,E2 -13518.092} C_VEL
LIN {X 0,Y 354.819,Z 732.289,A -85,B 0,C 180,E1 -13521.417,E2 -13521.417} C_VEL
LIN {X 0,Y 354.806,Z 732.286,A -85,B 0,C 180,E1 -13524.581,E2 -13524.581} C_VEL
LIN {X 0,Y 354.803,Z 732.286,A -85,B 0,C 180,E1 -13528.385,E2 -13528.385} C_VEL
LIN {X 0,Y 354.788,Z 732.289,A -85,B 0,C 180,E1 -13532.334,E2 -13532.334} C_VEL
LIN {X 0,Y 354.82,Z 732.289,A -85,B 0,C 180,E1 -13535.698,E2 -13535.698} C_VEL
LIN {X 0,Y 354.769,Z 732.294,A -85,B 0,C 180,E1 -13539.413,E2 -13539.413} C_VEL
LIN {X 0,Y 354.784,Z 732.289,A -85,B 0,C 180,E1 -13542.866,E2 -13542.866} C_VEL
LIN {X 0,Y 354.764,Z 732.296,A -85,B 0,C 180,E1 -13546.103,E2 -13546.103} C_VEL
LIN {X 0,Y 354.765,Z 732.291,A -85,B 0,C 180,E1 -13549.176,E2 -13549.176} C_VEL
LIN {X 0,Y 354.8,Z 732.29,A -85,B 0,C 180,E1 -13552.405,E2 -13552.405} C_VEL
LIN {X 0,Y 354.809,Z 732.286,A -85,B 0,C 180,E1 -13554.94,E2 -13554.94} C_VEL
LIN {X 0,Y 354.794,Z 732.292,A -85,B 0,C 180,E1 -13558.406,E2 -13558.406} C_VEL
LIN {X 0,Y 354.798,Z 732.287,A -85,B 0,C 180,E1 -13561.614,E2 -13561.614} C_VEL
LIN {X 0,Y 354.806,Z 732.286,A -85,B 0,C 180,E1 -13565.42,E2 -13565.42} C_VEL
LIN {X 0,Y 354.829,Z 732.285,A -85,B 0,C 180,E1 -13569.113,E2 -13569.113} C_VEL
LIN {X 0,Y 354.882,Z 732.281,A -85,B 0,C 180,E1 -13572.719,E2 -13572.719} C_VEL
LIN {X 0,Y 354.954,Z 732.269,A -85,B 0,C 180,E1 -13576.255,E2 -13576.255} C_VEL
LIN {X 0,Y 354.953,Z 732.268,A -85,B 0,C 180,E1 -13579.735,E2 -13579.735} C_VEL
LIN {X 0,Y 355.088,Z 732.255,A -85,B 0,C 180,E1 -13583.18,E2 -13583.18} C_VEL
LIN {X 0,Y 355.228,Z 732.234,A -85,B 0,C 180,E1 -13587.732,E2 -13587.732} C_VEL
LIN {X 0,Y 355.148,Z 732.248,A -85,B 0,C 180,E1 -13591.134,E2 -13591.134} C_VEL
